C09065=1103.745,273.305,-76.182,179.309,15.397,151.389
C09066=1103.739,273.056,-76.153,179.306,15.397,151.390
C09067=1103.734,272.808,-76.125,179.302,15.395,151.390
C09068=1103.728,272.560,-76.096,179.298,15.395,151.391
C09069=1103.723,272.312,-76.068,179.294,15.394,151.392
C09070=1103.717,272.063,-76.039,179.291,15.393,151.392
C09071=1103.711,271.815,-76.010,179.287,15.393,151.393
C09072=1103.706,271.567,-75.982,179.283,15.392,151.394
C09073=1103.700,271.318,-75.954,179.280,15.391,151.394
C09074=1103.695,271.070,-75.925,179.276,15.390,151.395
C09075=1103.689,270.822,-75.897,179.272,15.390,151.395
C09076=1103.683,270.574,-75.869,179.269,15.389,151.396
C09077=1103.677,270.325,-75.840,179.265,15.388,151.397
C09078=1103.671,270.077,-75.811,179.262,15.387,151.397
C09079=1103.666,269.829,-75.783,179.257,15.386,151.398
C09080=1103.660,269.580,-75.755,179.254,15.386,151.399
C09081=1103.655,269.332,-75.727,179.250,15.385,151.399
C09082=1103.649,269.083,-75.699,179.246,15.384,151.400
C09083=1103.644,268.835,-75.669,179.243,15.384,151.400
C09084=1103.638,268.587,-75.641,179.239,15.383,151.401
C09085=1103.632,268.339,-75.613,179.235,15.382,151.402
C09086=1103.626,268.090,-75.585,179.232,15.382,151.402
C09087=1103.621,267.842,-75.557,179.228,15.381,151.403
C09088=1103.615,267.593,-75.528,179.224,15.380,151.404
C09089=1103.610,267.345,-75.501,179.220,15.379,151.404
C09090=1103.604,267.097,-75.471,179.217,15.379,151.405
C09091=1103.598,266.849,-75.444,179.213,15.378,151.405
C09092=1103.592,266.600,-75.415,179.209,15.377,151.406
C09093=1103.587,266.352,-75.387,179.206,15.377,151.407
C09094=1103.581,266.103,-75.359,179.202,15.376,151.407
C09095=1103.576,265.855,-75.331,179.198,15.375,151.408
C09096=1103.570,265.606,-75.303,179.195,15.375,151.409
C09097=1103.564,265.358,-75.275,179.191,15.374,151.409
C09098=1103.558,265.110,-75.246,179.187,15.373,151.410
C09099=1103.552,264.862,-75.219,179.184,15.373,151.411
C09100=1103.547,264.614,-75.191,179.179,15.372,151.411
C09101=1103.541,264.365,-75.163,179.176,15.371,151.412
C09102=1103.536,264.117,-75.135,179.173,15.371,151.412
C09103=1103.530,263.868,-75.107,179.168,15.370,151.413
C09104=1103.525,263.620,-75.079,179.165,15.370,151.414
C09105=1103.516,263.267,-75.039,179.160,15.368,151.415
C09106=1103.507,262.913,-74.999,179.155,15.368,151.416
C09107=1103.499,262.559,-74.960,179.149,15.367,151.417
C09108=1103.491,262.206,-74.920,179.144,15.366,151.418
C09109=1103.486,261.957,-74.893,179.140,15.366,151.418
C09110=1103.480,261.708,-74.865,179.136,15.365,151.419
C09111=1103.475,261.460,-74.837,179.133,15.364,151.420
C09112=1103.468,261.212,-74.809,179.129,15.364,151.420
C09113=1103.463,260.964,-74.781,179.125,15.363,151.421
C09114=1103.458,260.715,-74.754,179.121,15.363,151.422
C09115=1103.451,260.467,-74.726,179.118,15.363,151.422
C09116=1103.445,260.219,-74.698,179.114,15.361,151.423
C09117=1103.440,259.970,-74.670,179.110,15.361,151.424
C09118=1103.434,259.721,-74.643,179.107,15.361,151.424
C09119=1103.428,259.473,-74.615,179.102,15.360,151.425
C09120=1103.422,259.225,-74.587,179.099,15.359,151.426
C09121=1103.417,258.976,-74.560,179.095,15.359,151.426
C09122=1103.411,258.728,-74.532,179.092,15.359,151.427
C09123=1103.405,258.480,-74.504,179.088,15.358,151.428
C09124=1103.400,258.231,-74.477,179.084,15.357,151.428
C09125=1103.394,257.982,-74.449,179.081,15.357,151.429
C09126=1103.389,257.734,-74.422,179.077,15.356,151.430
C09127=1103.383,257.486,-74.394,179.073,15.356,151.430
C09128=1103.377,257.237,-74.366,179.069,15.355,151.431
C09129=1103.371,256.989,-74.339,179.065,15.355,151.432
C09130=1103.366,256.741,-74.311,179.062,15.354,151.432
C09131=1103.360,256.492,-74.284,179.058,15.354,151.433
C09132=1103.354,256.244,-74.256,179.054,15.353,151.434
C09133=1103.349,255.995,-74.229,179.051,15.352,151.434
C09134=1103.343,255.747,-74.202,179.047,15.352,151.435
C09135=1103.337,255.498,-74.174,179.044,15.352,151.436
C09136=1103.332,255.250,-74.146,179.039,15.351,151.436
C09137=1103.326,255.002,-74.119,179.036,15.351,151.437
C09138=1103.321,254.753,-74.092,179.033,15.350,151.438
C09139=1103.314,254.504,-74.065,179.028,15.349,151.438
C09140=1103.309,254.256,-74.037,179.025,15.349,151.439
C09141=1103.303,254.008,-74.010,179.021,15.348,151.440
C09142=1103.298,253.759,-73.983,179.017,15.348,151.440
C09143=1103.292,253.510,-73.956,179.013,15.347,151.441
C09144=1103.286,253.262,-73.928,179.010,15.347,151.442
C09145=1103.281,253.014,-73.901,179.006,15.347,151.443
C09146=1103.276,252.765,-73.874,179.002,15.345,151.443
C09147=1103.269,252.517,-73.846,178.999,15.345,151.444
C09148=1103.264,252.268,-73.819,178.995,15.345,151.445
C09149=1103.258,252.020,-73.792,178.991,15.344,151.445
C09150=1103.253,251.772,-73.764,178.987,15.344,151.446
C09151=1103.247,251.523,-73.738,178.984,15.343,151.447
C09152=1103.242,251.275,-73.710,178.980,15.343,151.447
C09153=1103.236,251.026,-73.684,178.976,15.342,151.448
C09154=1103.230,250.778,-73.655,178.973,15.342,151.449
C09155=1103.224,250.529,-73.629,178.969,15.341,151.449
C09156=1103.219,250.280,-73.601,178.966,15.341,151.450
C09157=1103.211,249.924,-73.563,178.960,15.340,151.451
C09158=1103.203,249.568,-73.524,178.954,15.339,151.452
C09159=1103.195,249.212,-73.485,178.949,15.338,151.453
C09160=1103.187,248.854,-73.446,178.944,15.338,151.454
C09161=1103.182,248.606,-73.420,178.940,15.337,151.455
C09162=1103.176,248.358,-73.393,178.937,15.337,151.455
C09163=1103.171,248.110,-73.365,178.933,15.336,151.456
C09164=1103.165,247.861,-73.338,178.930,15.336,151.457
C09165=1103.160,247.613,-73.311,178.925,15.335,151.457
C09166=1103.154,247.364,-73.284,178.922,15.335,151.458
C09167=1103.148,247.116,-73.258,178.918,15.335,151.459
C09168=1103.142,246.868,-73.231,178.915,15.334,151.459
C09169=1103.137,246.619,-73.204,178.910,15.334,151.460
C09170=1103.131,246.370,-73.177,178.907,15.333,151.461
C09171=1103.125,246.121,-73.150,178.903,15.333,151.462
C09172=1103.120,245.873,-73.124,178.900,15.333,151.462
C09173=1103.114,245.624,-73.096,178.896,15.332,151.463
C09174=1103.109,245.376,-73.070,178.892,15.332,151.464
C09175=1103.103,245.128,-73.043,178.888,15.331,151.464
C09176=1103.097,244.879,-73.017,178.885,15.331,151.465
C09177=1103.092,244.630,-72.990,178.881,15.331,151.466
C09178=1103.087,244.382,-72.963,178.877,15.330,151.466
C09179=1103.081,244.133,-72.937,178.874,15.330,151.467
C09180=1103.075,243.885,-72.910,178.870,15.329,151.468
C09181=1103.069,243.637,-72.883,178.867,15.329,151.469
C09182=1103.064,243.388,-72.856,178.862,15.328,151.469
C09183=1103.059,243.139,-72.830,178.859,15.328,151.470
C09184=1103.053,242.891,-72.804,178.855,15.328,151.471
C09185=1103.046,242.576,-72.770,178.851,15.327,151.472
C09186=1103.038,242.261,-72.736,178.846,15.327,151.473
C09187=1103.031,241.946,-72.703,178.841,15.327,151.473
C09188=1103.023,241.631,-72.669,178.836,15.326,151.474
C09189=1103.018,241.382,-72.643,178.832,15.325,151.475
C09190=1103.012,241.133,-72.616,178.829,15.325,151.476
C09191=1103.006,240.885,-72.589,178.825,15.325,151.476
C09192=1103.001,240.637,-72.563,178.821,15.325,151.477
C09193=1102.996,240.387,-72.536,178.818,15.324,151.478
C09194=1102.990,240.139,-72.510,178.813,15.324,151.479
C09195=1102.984,239.891,-72.483,178.810,15.324,151.479
C09196=1102.978,239.642,-72.458,178.806,15.323,151.480
C09197=1102.972,239.394,-72.431,178.803,15.323,151.481
C09198=1102.966,239.145,-72.404,178.799,15.323,151.482
C09199=1102.961,238.896,-72.378,178.795,15.322,151.482
C09200=1102.955,238.648,-72.352,178.791,15.322,151.483
C09201=1102.950,238.399,-72.326,178.788,15.321,151.484
C09202=1102.944,238.151,-72.299,178.784,15.321,151.484
C09203=1102.938,237.902,-72.273,178.780,15.321,151.485
C09204=1102.933,237.653,-72.247,178.777,15.321,151.486
C09205=1102.927,237.405,-72.220,178.773,15.320,151.487
C09206=1102.922,237.157,-72.194,178.769,15.320,151.487
C09207=1102.916,236.908,-72.168,178.766,15.320,151.488
C09208=1102.911,236.659,-72.142,178.762,15.320,151.489
C09209=1102.904,236.362,-72.111,178.757,15.319,151.490
C09210=1102.896,236.066,-72.079,178.753,15.319,151.491
C09211=1102.891,235.769,-72.048,178.748,15.318,151.491
C09212=1102.884,235.472,-72.017,178.744,15.318,151.492
C09213=1102.878,235.224,-71.990,178.740,15.317,151.493
C09214=1102.872,234.975,-71.964,178.736,15.317,151.494
C09215=1102.867,234.727,-71.939,178.733,15.317,151.494
C09216=1102.861,234.479,-71.913,178.729,15.317,151.495
C09217=1102.856,234.230,-71.887,178.726,15.316,151.496
C09218=1102.850,233.981,-71.861,178.722,15.317,151.497
C09219=1102.844,233.732,-71.834,178.718,15.316,151.497
C09220=1102.839,233.483,-71.808,178.714,15.316,151.498
C09221=1102.833,233.235,-71.783,178.711,15.315,151.499
C09222=1102.827,232.987,-71.757,178.707,15.315,151.500
C09223=1102.822,232.738,-71.731,178.704,15.315,151.500
C09224=1102.817,232.489,-71.705,178.700,15.315,151.501
C09225=1102.810,232.241,-71.679,178.695,15.314,151.502
C09226=1102.805,231.992,-71.653,178.692,15.314,151.503
C09227=1102.799,231.743,-71.627,178.688,15.314,151.503
C09228=1102.794,231.495,-71.601,178.685,15.313,151.504
C09229=1102.788,231.247,-71.575,178.681,15.313,151.505
C09230=1102.782,230.998,-71.549,178.678,15.313,151.505
C09231=1102.777,230.749,-71.523,178.674,15.313,151.506
C09232=1102.771,230.500,-71.498,178.670,15.312,151.507
C09233=1102.766,230.252,-71.472,178.666,15.312,151.508
C09234=1102.760,230.003,-71.446,178.662,15.312,151.508
C09235=1102.754,229.755,-71.420,178.659,15.312,151.509
C09236=1102.748,229.506,-71.394,178.655,15.312,151.510
C09237=1102.742,229.257,-71.369,178.651,15.312,151.511
C09238=1102.737,229.009,-71.344,178.648,15.311,151.511
C09239=1102.732,228.760,-71.318,178.644,15.311,151.512
C09240=1102.725,228.511,-71.292,178.640,15.311,151.513
C09241=1102.720,228.262,-71.266,178.636,15.310,151.514
C09242=1102.714,228.013,-71.241,178.633,15.310,151.514
C09243=1102.709,227.765,-71.215,178.629,15.310,151.515
C09244=1102.703,227.517,-71.190,178.625,15.310,151.516
C09245=1102.697,227.268,-71.164,178.622,15.310,151.517
C09246=1102.691,227.019,-71.139,178.618,15.310,151.517
C09247=1102.686,226.771,-71.113,178.615,15.310,151.518
C09248=1102.680,226.522,-71.088,178.610,15.309,151.519
C09249=1102.675,226.273,-71.062,178.607,15.309,151.520
C09250=1102.669,226.025,-71.037,178.603,15.309,151.520
C09251=1102.663,225.776,-71.011,178.599,15.308,151.521
C09252=1102.657,225.527,-70.986,178.596,15.308,151.522
C09253=1102.652,225.278,-70.960,178.592,15.308,151.523
C09254=1102.646,225.030,-70.935,178.588,15.308,151.523
C09255=1102.641,224.781,-70.909,178.585,15.308,151.524
C09256=1102.634,224.533,-70.884,178.581,15.308,151.525
C09257=1102.630,224.284,-70.858,178.577,15.307,151.526
C09258=1102.623,224.036,-70.833,178.573,15.307,151.527
C09259=1102.618,223.787,-70.807,178.570,15.307,151.527
C09260=1102.613,223.538,-70.783,178.566,15.307,151.528
C09261=1102.604,223.166,-70.744,178.560,15.306,151.529
C09262=1102.596,222.795,-70.706,178.555,15.306,151.530
C09263=1102.587,222.424,-70.669,178.550,15.306,151.531
C09264=1102.579,222.051,-70.631,178.545,15.306,151.532
C09265=1102.574,221.803,-70.606,178.540,15.305,151.533
C09266=1102.567,221.555,-70.580,178.536,15.305,151.534
C09267=1102.562,221.305,-70.555,178.533,15.305,151.535
C09268=1102.557,221.057,-70.530,178.529,15.305,151.535
C09269=1102.550,220.809,-70.505,178.525,15.305,151.536
C09270=1102.545,220.560,-70.479,178.522,15.305,151.537
C09271=1102.540,220.311,-70.455,178.518,15.304,151.538
C09272=1102.533,220.062,-70.429,178.514,15.305,151.539
C09273=1102.527,219.814,-70.404,178.511,15.305,151.539
C09274=1102.523,219.565,-70.379,178.507,15.304,151.540
C09275=1102.516,219.316,-70.354,178.504,15.304,151.541
C09276=1102.511,219.068,-70.330,178.500,15.304,151.542
C09277=1102.505,218.819,-70.304,178.496,15.304,151.542
C09278=1102.499,218.570,-70.278,178.493,15.304,151.543
C09279=1102.494,218.321,-70.254,178.488,15.303,151.544
C09280=1102.488,218.073,-70.229,178.485,15.303,151.545
C09281=1102.483,217.824,-70.204,178.481,15.303,151.545
C09282=1102.476,217.575,-70.179,178.478,15.303,151.546
C09283=1102.472,217.326,-70.154,178.474,15.303,151.547
C09284=1102.466,217.078,-70.129,178.470,15.303,151.548
C09285=1102.460,216.829,-70.105,178.467,15.303,151.548
C09286=1102.454,216.581,-70.079,178.463,15.303,151.549
C09287=1102.449,216.332,-70.055,178.459,15.303,151.550
C09288=1102.443,216.083,-70.029,178.456,15.302,151.551
C09289=1102.438,215.834,-70.005,178.452,15.302,151.551
C09290=1102.432,215.586,-69.979,178.448,15.302,151.552
C09291=1102.427,215.337,-69.955,178.445,15.302,151.553
C09292=1102.420,215.088,-69.930,178.441,15.302,151.554
C09293=1102.415,214.840,-69.906,178.438,15.302,151.554
C09294=1102.409,214.591,-69.880,178.434,15.302,151.555
C09295=1102.404,214.342,-69.855,178.430,15.302,151.556
C09296=1102.398,214.093,-69.831,178.426,15.301,151.557
C09297=1102.393,213.845,-69.806,178.422,15.301,151.558
C09298=1102.387,213.596,-69.781,178.419,15.301,151.558
C09299=1102.382,213.347,-69.757,178.415,15.301,151.559
C09300=1102.375,213.098,-69.732,178.411,15.301,151.560
C09301=1102.370,212.850,-69.707,178.408,15.301,151.561
C09302=1102.364,212.601,-69.683,178.404,15.301,151.561
C09303=1102.359,212.353,-69.658,178.400,15.301,151.562
C09304=1102.353,212.103,-69.633,178.397,15.301,151.563
C09305=1102.347,211.855,-69.609,178.393,15.301,151.564
C09306=1102.342,211.606,-69.585,178.390,15.300,151.564
C09307=1102.336,211.358,-69.559,178.386,15.301,151.565
C09308=1102.331,211.109,-69.535,178.382,15.300,151.566
C09309=1102.325,210.860,-69.510,178.379,15.300,151.567
C09310=1102.319,210.611,-69.486,178.375,15.300,151.568
C09311=1102.313,210.362,-69.461,178.371,15.300,151.568
C09312=1102.308,210.114,-69.437,178.368,15.300,151.569
C09313=1102.299,209.746,-69.401,178.362,15.300,151.570
C09314=1102.291,209.378,-69.364,178.357,15.300,151.571
C09315=1102.283,209.010,-69.329,178.352,15.300,151.572
C09316=1102.274,208.642,-69.292,178.346,15.300,151.574
C09317=1102.252,207.639,-69.194,178.312,15.293,151.579
C09318=1102.246,207.391,-69.170,178.308,15.294,151.580
C09319=1102.240,207.142,-69.146,178.304,15.294,151.581
C09320=1102.234,206.893,-69.122,178.301,15.296,151.582
C09321=1102.229,206.644,-69.097,178.297,15.296,151.583
C09322=1102.222,206.395,-69.073,178.292,15.297,151.585
C09323=1102.217,206.147,-69.049,178.289,15.297,151.585
C09324=1102.212,205.898,-69.025,178.285,15.299,151.586
C09325=1102.206,205.648,-69.001,178.281,15.299,151.587
C09326=1102.200,205.400,-68.977,178.277,15.300,151.589
C09327=1102.195,205.151,-68.953,178.274,15.301,151.589
C09328=1102.190,204.903,-68.929,178.269,15.302,151.590
C09329=1102.183,204.654,-68.905,178.265,15.302,151.591
C09330=1102.178,204.405,-68.880,178.261,15.303,151.593
C09331=1102.172,204.157,-68.856,178.258,15.304,151.593
C09332=1102.167,203.908,-68.833,178.254,15.305,151.594
C09333=1102.161,203.659,-68.809,178.250,15.305,151.596
C09334=1102.155,203.410,-68.784,178.246,15.305,151.596
C09335=1102.149,203.162,-68.761,178.242,15.307,151.597
C09336=1102.144,202.913,-68.736,178.238,15.307,151.598
C09337=1102.139,202.663,-68.712,178.234,15.308,151.600
C09338=1102.132,202.415,-68.689,178.231,15.309,151.600
C09339=1102.127,202.166,-68.665,178.227,15.310,151.601
C09340=1102.121,201.917,-68.641,178.222,15.310,151.603
C09341=1102.116,201.668,-68.617,178.218,15.311,151.604
C09342=1102.110,201.420,-68.593,178.215,15.312,151.604
C09343=1102.104,201.171,-68.569,178.211,15.313,151.605
C09344=1102.098,200.922,-68.545,178.207,15.314,151.607
C09345=1102.093,200.673,-68.521,178.203,15.315,151.608
C09346=1102.087,200.425,-68.498,178.200,15.315,151.608
C09347=1102.081,200.177,-68.474,178.195,15.316,151.610
C09348=1102.075,199.927,-68.450,178.191,15.317,151.611
C09349=1102.069,199.678,-68.427,178.188,15.317,151.611
C09350=1102.064,199.430,-68.402,178.184,15.318,151.612
C09351=1102.058,199.181,-68.379,178.180,15.319,151.614
C09352=1102.052,198.932,-68.355,178.177,15.320,151.614
C09353=1102.046,198.683,-68.332,178.172,15.320,151.615
C09354=1102.041,198.434,-68.308,178.168,15.321,151.617
C09355=1102.035,198.185,-68.285,178.165,15.322,151.617
C09356=1102.029,197.937,-68.261,178.161,15.323,151.618
C09357=1102.023,197.688,-68.236,178.157,15.323,151.620
C09358=1102.018,197.439,-68.213,178.153,15.324,151.620
C09359=1102.012,197.190,-68.189,178.149,15.325,151.621
C09360=1102.006,196.941,-68.166,178.146,15.325,151.622
C09361=1102.000,196.693,-68.143,178.141,15.326,151.623
C09362=1101.995,196.444,-68.119,178.138,15.327,151.624
C09363=1101.989,196.195,-68.095,178.134,15.328,151.625
C09364=1101.983,195.946,-68.072,178.130,15.328,151.626
C09365=1101.978,195.697,-68.048,178.127,15.329,151.627
C09366=1101.972,195.448,-68.025,178.123,15.330,151.628
C09367=1101.966,195.199,-68.002,178.119,15.330,151.629
C09368=1101.961,194.951,-67.978,178.115,15.331,151.630
C09369=1101.955,194.702,-67.955,178.111,15.332,151.631
C09370=1101.949,194.454,-67.931,178.107,15.333,151.632
C09371=1101.944,194.204,-67.907,178.103,15.333,151.633
C09372=1101.938,193.955,-67.884,178.100,15.334,151.634
C09373=1101.932,193.707,-67.860,178.096,15.335,151.635
C09374=1101.927,193.457,-67.837,178.092,15.335,151.636
C09375=1101.921,193.209,-67.814,178.089,15.336,151.637
C09376=1101.915,192.960,-67.790,178.085,15.337,151.638
C09377=1101.910,192.711,-67.767,178.081,15.337,151.639
C09378=1101.904,192.439,-67.742,178.077,15.338,151.640
C09379=1101.897,192.167,-67.715,178.072,15.339,151.641
C09380=1101.892,191.894,-67.690,178.068,15.339,151.642
C09381=1101.885,191.621,-67.665,178.064,15.340,151.643
C09382=1101.879,191.373,-67.642,178.061,15.342,151.644
C09383=1101.874,191.123,-67.618,178.057,15.342,151.645
C09384=1101.868,190.875,-67.595,178.053,15.342,151.646
C09385=1101.862,190.626,-67.572,178.049,15.344,151.647
C09386=1101.857,190.377,-67.549,178.046,15.344,151.648
C09387=1101.852,190.128,-67.525,178.041,15.345,151.649
C09388=1101.846,189.879,-67.502,178.037,15.345,151.650
C09389=1101.840,189.631,-67.479,178.034,15.346,151.651
C09390=1101.834,189.382,-67.456,178.030,15.346,151.652
C09391=1101.829,189.133,-67.432,178.026,15.347,151.653
C09392=1101.823,188.884,-67.409,178.023,15.348,151.653
C09393=1101.818,188.635,-67.386,178.019,15.348,151.655
C09394=1101.812,188.386,-67.363,178.015,15.349,151.655
C09395=1101.807,188.138,-67.341,178.012,15.350,151.656
C09396=1101.802,187.889,-67.317,178.008,15.350,151.657
C09397=1101.796,187.640,-67.294,178.004,15.351,151.658
C09398=1101.790,187.392,-67.271,178.001,15.352,151.659
C09399=1101.784,187.143,-67.248,177.997,15.352,151.660
C09400=1101.779,186.894,-67.225,177.993,15.353,151.661
C09401=1101.774,186.645,-67.201,177.989,15.353,151.662
C09402=1101.768,186.396,-67.178,177.986,15.354,151.663
C09403=1101.762,186.147,-67.155,177.982,15.354,151.664
C09404=1101.756,185.898,-67.132,177.978,15.355,151.665
C09405=1101.751,185.649,-67.109,177.975,15.356,151.666
C09406=1101.746,185.401,-67.087,177.971,15.356,151.667
C09407=1101.740,185.152,-67.064,177.967,15.357,151.667
C09408=1101.734,184.902,-67.042,177.963,15.358,151.668
C09409=1101.729,184.653,-67.019,177.960,15.358,151.669
C09410=1101.723,184.405,-66.996,177.956,15.358,151.670
C09411=1101.717,184.156,-66.973,177.952,15.360,151.671
C09412=1101.712,183.907,-66.950,177.948,15.360,151.672
C09413=1101.706,183.658,-66.927,177.945,15.360,151.673
C09414=1101.700,183.409,-66.904,177.941,15.362,151.674
C09415=1101.694,183.160,-66.882,177.937,15.362,151.675
C09416=1101.688,182.912,-66.859,177.933,15.362,151.676
C09417=1101.682,182.663,-66.836,177.930,15.364,151.677
C09418=1101.676,182.414,-66.813,177.926,15.364,151.678
C09419=1101.671,182.164,-66.791,177.922,15.364,151.679
C09420=1101.665,181.915,-66.768,177.919,15.366,151.680
C09421=1101.659,181.667,-66.745,177.915,15.366,151.681
C09422=1101.653,181.418,-66.722,177.911,15.367,151.682
C09423=1101.647,181.169,-66.699,177.908,15.367,151.682
C09424=1101.642,180.919,-66.677,177.904,15.368,151.684
C09425=1101.636,180.670,-66.654,177.900,15.369,151.684
C09426=1101.630,180.423,-66.632,177.897,15.369,151.685
C09427=1101.625,180.174,-66.609,177.893,15.370,151.686
C09428=1101.619,179.924,-66.587,177.889,15.371,151.687
C09429=1101.613,179.675,-66.564,177.886,15.371,151.688
C09430=1101.608,179.426,-66.541,177.882,15.372,151.689
C09431=1101.601,179.178,-66.519,177.878,15.372,151.690
C09432=1101.596,178.928,-66.497,177.875,15.373,151.691
C09433=1101.590,178.679,-66.474,177.871,15.374,151.692
C09434=1101.585,178.431,-66.451,177.867,15.374,151.693
C09435=1101.579,178.182,-66.429,177.864,15.375,151.694
C09436=1101.573,177.933,-66.406,177.860,15.375,151.695
C09437=1101.567,177.684,-66.384,177.856,15.376,151.695
C09438=1101.562,177.435,-66.361,177.853,15.377,151.696
C09439=1101.555,177.186,-66.339,177.849,15.377,151.697
C09440=1101.551,176.937,-66.317,177.845,15.378,151.698
C09441=1101.545,176.688,-66.294,177.842,15.379,151.699
C09442=1101.539,176.415,-66.270,177.838,15.379,151.700
C09443=1101.532,176.143,-66.245,177.833,15.380,151.701
C09444=1101.526,175.870,-66.221,177.830,15.380,151.702
C09445=1101.519,175.597,-66.196,177.825,15.381,151.703
C09446=1101.514,175.349,-66.174,177.822,15.382,151.704
C09447=1101.509,175.099,-66.151,177.818,15.382,151.705
C09448=1101.502,174.851,-66.129,177.815,15.383,151.706
C09449=1101.497,174.601,-66.107,177.811,15.384,151.707
C09450=1101.492,174.353,-66.084,177.808,15.384,151.707
C09451=1101.486,174.104,-66.063,177.804,15.384,151.708
C09452=1101.480,173.855,-66.040,177.801,15.385,151.709
C09453=1101.474,173.605,-66.017,177.797,15.385,151.710
C09454=1101.469,173.357,-65.995,177.793,15.386,151.711
C09455=1101.463,173.108,-65.973,177.790,15.387,151.712
C09456=1101.457,172.859,-65.952,177.786,15.387,151.713
C09457=1101.452,172.611,-65.929,177.782,15.387,151.714
C09458=1101.446,172.361,-65.907,177.779,15.388,151.715
C09459=1101.440,172.112,-65.884,177.775,15.389,151.715
C09460=1101.435,171.863,-65.862,177.771,15.389,151.716
C09461=1101.430,171.614,-65.840,177.768,15.390,151.717
C09462=1101.423,171.366,-65.818,177.764,15.390,151.718
C09463=1101.418,171.116,-65.796,177.761,15.390,151.719
C09464=1101.412,170.867,-65.775,177.757,15.391,151.720
C09465=1101.407,170.619,-65.752,177.754,15.392,151.721
C09466=1101.401,170.369,-65.729,177.750,15.392,151.722
C09467=1101.396,170.121,-65.708,177.747,15.393,151.722
C09468=1101.390,169.872,-65.685,177.743,15.393,151.723
C09469=1101.384,169.622,-65.663,177.740,15.394,151.724
C09470=1101.379,169.374,-65.642,177.736,15.394,151.725
C09471=1101.373,169.124,-65.620,177.732,15.394,151.726
C09472=1101.368,168.876,-65.597,177.729,15.395,151.727
C09473=1101.362,168.627,-65.575,177.725,15.396,151.728
C09474=1101.356,168.378,-65.554,177.721,15.396,151.729
C09475=1101.351,168.129,-65.532,177.718,15.397,151.729
C09476=1101.345,167.880,-65.510,177.715,15.397,151.730
C09477=1101.340,167.631,-65.487,177.711,15.397,151.731
C09478=1101.334,167.382,-65.466,177.708,15.398,151.732
C09479=1101.328,167.133,-65.444,177.704,15.398,151.733
C09480=1101.323,166.884,-65.422,177.700,15.398,151.734
C09481=1101.317,166.635,-65.400,177.697,15.399,151.734
C09482=1101.312,166.386,-65.379,177.693,15.400,151.735
C09483=1101.306,166.137,-65.357,177.690,15.400,151.736
C09484=1101.301,165.888,-65.335,177.687,15.401,151.737
C09485=1101.295,165.639,-65.312,177.683,15.401,151.738
C09486=1101.289,165.391,-65.291,177.680,15.402,151.739
C09487=1101.284,165.141,-65.269,177.676,15.402,151.739
C09488=1101.278,164.893,-65.248,177.672,15.402,151.740
C09489=1101.273,164.643,-65.225,177.669,15.403,151.741
C09490=1101.267,164.394,-65.204,177.665,15.403,151.742
C09491=1101.262,164.145,-65.182,177.662,15.403,151.743
C09492=1101.256,163.896,-65.160,177.659,15.404,151.744
C09493=1101.251,163.647,-65.138,177.655,15.404,151.745
C09494=1101.245,163.399,-65.117,177.651,15.405,151.745
C09495=1101.239,163.149,-65.095,177.648,15.405,151.746
C09496=1101.235,162.901,-65.074,177.644,15.406,151.747
C09497=1101.228,162.651,-65.052,177.641,15.406,151.748
C09498=1101.224,162.403,-65.030,177.638,15.406,151.749
C09499=1101.217,162.153,-65.008,177.634,15.406,151.749
C09500=1101.213,161.905,-64.987,177.631,15.407,151.750
C09501=1101.207,161.655,-64.966,177.627,15.408,151.751
C09502=1101.201,161.406,-64.944,177.624,15.408,151.752
C09503=1101.195,161.157,-64.923,177.620,15.409,151.753
C09504=1101.190,160.908,-64.901,177.617,15.409,151.754
C09505=1101.184,160.659,-64.879,177.613,15.409,151.754
C09506=1101.178,160.385,-64.856,177.610,15.410,151.755
C09507=1101.172,160.113,-64.832,177.606,15.410,151.756
C09508=1101.166,159.840,-64.809,177.602,15.411,151.757
C09509=1101.159,159.567,-64.785,177.598,15.411,151.758
C09510=1101.154,159.318,-64.764,177.594,15.411,151.759
C09511=1101.148,159.068,-64.742,177.591,15.412,151.760
C09512=1101.142,158.820,-64.721,177.588,15.412,151.761
C09513=1101.136,158.571,-64.699,177.584,15.413,151.761
C09514=1101.131,158.322,-64.678,177.581,15.413,151.762
C09515=1101.125,158.072,-64.657,177.577,15.413,151.763
C09516=1101.120,157.823,-64.635,177.574,15.414,151.764
C09517=1101.114,157.574,-64.614,177.570,15.414,151.765
C09518=1101.108,157.326,-64.592,177.567,15.414,151.765
C09519=1101.102,157.076,-64.572,177.564,15.415,151.766
C09520=1101.097,156.827,-64.550,177.560,15.415,151.767
C09521=1101.091,156.579,-64.529,177.556,15.416,151.768
C09522=1101.085,156.329,-64.508,177.554,15.416,151.769
C09523=1101.080,156.080,-64.486,177.550,15.417,151.770
C09524=1101.074,155.831,-64.465,177.547,15.417,151.770
C09525=1101.069,155.582,-64.444,177.543,15.417,151.771
C09526=1101.064,155.333,-64.423,177.539,15.417,151.772
C09527=1101.057,155.084,-64.401,177.536,15.418,151.773
C09528=1101.052,154.835,-64.381,177.533,15.418,151.774
C09529=1101.046,154.586,-64.359,177.530,15.419,151.774
C09530=1101.040,154.337,-64.338,177.526,15.419,151.775
C09531=1101.035,154.088,-64.317,177.522,15.420,151.776
C09532=1101.029,153.839,-64.295,177.519,15.420,151.777
C09533=1101.024,153.590,-64.275,177.515,15.420,151.778
C09534=1101.018,153.341,-64.253,177.512,15.420,151.778
C09535=1101.012,153.092,-64.232,177.509,15.421,151.779
C09536=1101.007,152.843,-64.211,177.505,15.421,151.780
C09537=1101.001,152.594,-64.190,177.502,15.422,151.781
C09538=1100.995,152.345,-64.169,177.499,15.422,151.782
C09539=1100.989,152.096,-64.148,177.495,15.422,151.782
C09540=1100.984,151.846,-64.127,177.492,15.423,151.783
C09541=1100.978,151.598,-64.106,177.488,15.423,151.784
C09542=1100.972,151.348,-64.085,177.486,15.424,151.785
C09543=1100.967,151.100,-64.064,177.482,15.424,151.786
C09544=1100.962,150.851,-64.043,177.478,15.424,151.786
C09545=1100.955,150.601,-64.021,177.475,15.425,151.787
C09546=1100.950,150.352,-64.001,177.472,15.424,151.788
C09547=1100.945,150.103,-63.980,177.469,15.425,151.789
C09548=1100.939,149.854,-63.959,177.465,15.425,151.790
C09549=1100.933,149.605,-63.939,177.461,15.425,151.790
C09550=1100.927,149.357,-63.917,177.459,15.426,151.791
C09551=1100.922,149.107,-63.897,177.455,15.426,151.792
C09552=1100.916,148.858,-63.876,177.452,15.427,151.793
C09553=1100.911,148.609,-63.855,177.448,15.427,151.793
C09554=1100.905,148.360,-63.834,177.445,15.427,151.794
C09555=1100.899,148.110,-63.813,177.442,15.428,151.795
C09556=1100.894,147.862,-63.792,177.438,15.428,151.796
C09557=1100.888,147.613,-63.772,177.435,15.428,151.796
C09558=1100.882,147.363,-63.751,177.431,15.429,151.797
C09559=1100.876,147.114,-63.730,177.428,15.429,151.798
C09560=1100.871,146.865,-63.709,177.425,15.429,151.799
C09561=1100.865,146.617,-63.689,177.422,15.429,151.800
C09562=1100.859,146.367,-63.668,177.418,15.430,151.800
C09563=1100.854,146.118,-63.647,177.415,15.430,151.801
C09564=1100.849,145.869,-63.627,177.411,15.430,151.802
C09565=1100.842,145.620,-63.606,177.408,15.430,151.803
C09566=1100.836,145.371,-63.585,177.405,15.430,151.803
C09567=1100.831,145.122,-63.564,177.402,15.431,151.804
C09568=1100.826,144.873,-63.544,177.398,15.431,151.805
C09569=1100.820,144.624,-63.524,177.395,15.431,151.806
C09570=1100.814,144.350,-63.500,177.392,15.432,151.807
C09571=1100.807,144.076,-63.478,177.388,15.432,151.807
C09572=1100.801,143.804,-63.455,177.384,15.433,151.808
C09573=1100.795,143.530,-63.433,177.381,15.433,151.809
C09574=1100.789,143.281,-63.412,177.377,15.433,151.810
C09575=1100.784,143.032,-63.391,177.374,15.433,151.810
C09576=1100.778,142.783,-63.371,177.371,15.433,151.811
C09577=1100.772,142.534,-63.351,177.368,15.434,151.812
C09578=1100.767,142.284,-63.330,177.364,15.434,151.813
C09579=1100.761,142.036,-63.310,177.361,15.435,151.814
C09580=1100.756,141.787,-63.289,177.358,15.434,151.814
C09581=1100.751,141.537,-63.269,177.354,15.434,151.815
C09582=1100.745,141.289,-63.249,177.351,15.435,151.816
C09583=1100.739,141.039,-63.228,177.348,15.435,151.817
C09584=1100.733,140.790,-63.207,177.345,15.436,151.817
C09585=1100.727,140.541,-63.187,177.341,15.435,151.818
C09586=1100.722,140.292,-63.166,177.338,15.435,151.819
C09587=1100.716,140.044,-63.146,177.335,15.436,151.819
C09588=1100.711,139.794,-63.126,177.331,15.436,151.820
C09589=1100.705,139.545,-63.105,177.329,15.436,151.821
C09590=1100.699,139.295,-63.086,177.325,15.436,151.822
C09591=1100.694,139.046,-63.065,177.321,15.436,151.822
C09592=1100.688,138.797,-63.045,177.319,15.437,151.823
C09593=1100.683,138.548,-63.024,177.315,15.437,151.824
C09594=1100.677,138.299,-63.005,177.312,15.437,151.825
C09595=1100.671,138.050,-62.984,177.309,15.437,151.825
C09596=1100.665,137.801,-62.964,177.306,15.438,151.826
C09597=1100.659,137.551,-62.943,177.302,15.438,151.827
C09598=1100.653,137.303,-62.923,177.299,15.438,151.828
C09599=1100.648,137.054,-62.903,177.296,15.438,151.828
C09600=1100.642,136.805,-62.883,177.292,15.438,151.829
C09601=1100.637,136.556,-62.862,177.290,15.439,151.830
C09602=1100.631,136.306,-62.843,177.286,15.439,151.831
C09603=1100.626,136.057,-62.822,177.283,15.439,151.831
C09604=1100.620,135.808,-62.802,177.280,15.439,151.832
C09605=1100.614,135.558,-62.781,177.276,15.439,151.833
C09606=1100.608,135.310,-62.761,177.274,15.440,151.833
C09607=1100.603,135.060,-62.741,177.270,15.440,151.834
C09608=1100.597,134.811,-62.722,177.267,15.440,151.835
C09609=1100.592,134.562,-62.701,177.264,15.440,151.835
C09610=1100.586,134.313,-62.681,177.261,15.441,151.836
C09611=1100.580,134.064,-62.661,177.257,15.440,151.837
C09612=1100.575,133.815,-62.641,177.254,15.440,151.838
C09613=1100.569,133.566,-62.621,177.251,15.441,151.838
C09614=1100.564,133.317,-62.601,177.248,15.441,151.839
C09615=1100.558,133.068,-62.581,177.245,15.441,151.840
C09616=1100.552,132.818,-62.562,177.241,15.441,151.840
C09617=1100.547,132.569,-62.541,177.239,15.441,151.841
C09618=1100.541,132.320,-62.521,177.235,15.441,151.842
C09619=1100.536,132.071,-62.501,177.232,15.441,151.843
C09620=1100.530,131.822,-62.481,177.229,15.442,151.843
C09621=1100.524,131.573,-62.461,177.225,15.441,151.844
C09622=1100.518,131.324,-62.442,177.223,15.442,151.845
C09623=1100.513,131.074,-62.422,177.219,15.442,151.845
C09624=1100.506,130.825,-62.401,177.216,15.442,151.846
C09625=1100.501,130.576,-62.382,177.213,15.442,151.847
C09626=1100.495,130.327,-62.362,177.210,15.443,151.848
C09627=1100.489,130.078,-62.342,177.207,15.442,151.848
C09628=1100.484,129.828,-62.322,177.203,15.442,151.849
C09629=1100.478,129.579,-62.302,177.200,15.443,151.850
C09630=1100.472,129.330,-62.283,177.197,15.443,151.850
C09631=1100.466,129.081,-62.263,177.194,15.443,151.851
C09632=1100.460,128.832,-62.243,177.191,15.443,151.852
C09633=1100.455,128.583,-62.223,177.188,15.444,151.852
C09634=1100.449,128.310,-62.202,177.184,15.444,151.853
C09635=1100.443,128.036,-62.180,177.181,15.444,151.854
C09636=1100.436,127.763,-62.158,177.177,15.444,151.855
C09637=1100.430,127.489,-62.137,177.174,15.444,151.855
C09638=1100.424,127.240,-62.117,177.171,15.444,151.856
C09639=1100.418,126.991,-62.098,177.167,15.444,151.857
C09640=1100.413,126.741,-62.077,177.165,15.444,151.857
C09641=1100.407,126.492,-62.058,177.161,15.444,151.858
C09642=1100.401,126.243,-62.038,177.159,15.444,151.859
C09643=1100.396,125.994,-62.019,177.155,15.444,151.859
C09644=1100.390,125.745,-61.999,177.152,15.445,151.860
C09645=1100.384,125.496,-61.980,177.149,15.444,151.861
C09646=1100.378,125.246,-61.961,177.145,15.444,151.862
C09647=1100.372,124.997,-61.941,177.143,15.445,151.862
C09648=1100.367,124.748,-61.921,177.139,15.444,151.863
C09649=1100.361,124.499,-61.901,177.137,15.445,151.864
C09650=1100.356,124.250,-61.882,177.133,15.445,151.864
C09651=1100.351,124.001,-61.863,177.130,15.445,151.865
C09652=1100.345,123.752,-61.843,177.127,15.445,151.865
C09653=1100.339,123.502,-61.823,177.124,15.445,151.866
C09654=1100.333,123.253,-61.804,177.121,15.445,151.867
C09655=1100.327,123.004,-61.784,177.118,15.445,151.867
C09656=1100.322,122.755,-61.765,177.115,15.445,151.868
C09657=1100.316,122.505,-61.746,177.112,15.445,151.869
C09658=1100.312,122.256,-61.726,177.109,15.445,151.869
C09659=1100.306,122.007,-61.706,177.105,15.445,151.870
C09660=1100.300,121.758,-61.687,177.103,15.445,151.871
C09661=1100.294,121.509,-61.668,177.099,15.445,151.871
C09662=1100.288,121.260,-61.648,177.097,15.445,151.872
C09663=1100.283,121.010,-61.629,177.093,15.445,151.873
C09664=1100.277,120.761,-61.609,177.091,15.445,151.873
C09665=1100.272,120.512,-61.591,177.087,15.445,151.874
C09666=1100.266,120.263,-61.571,177.085,15.445,151.875
C09667=1100.260,120.014,-61.551,177.082,15.445,151.875
C09668=1100.254,119.764,-61.532,177.078,15.445,151.876
C09669=1100.249,119.515,-61.513,177.075,15.445,151.877
C09670=1100.244,119.266,-61.494,177.072,15.445,151.877
C09671=1100.238,119.017,-61.475,177.069,15.445,151.878
C09672=1100.232,118.767,-61.455,177.066,15.445,151.878
C09673=1100.226,118.519,-61.436,177.063,15.445,151.879
C09674=1100.221,118.270,-61.417,177.060,15.445,151.880
C09675=1100.216,118.020,-61.397,177.058,15.445,151.880
C09676=1100.210,117.771,-61.378,177.054,15.445,151.881
C09677=1100.204,117.522,-61.359,177.051,15.445,151.882
C09678=1100.198,117.272,-61.340,177.048,15.445,151.882
C09679=1100.193,117.023,-61.321,177.045,15.445,151.883
C09680=1100.188,116.774,-61.302,177.042,15.445,151.884
C09681=1100.182,116.525,-61.282,177.039,15.444,151.884
C09682=1100.177,116.276,-61.263,177.036,15.444,151.885
C09683=1100.171,116.026,-61.244,177.033,15.444,151.885
C09684=1100.166,115.777,-61.225,177.030,15.445,151.886
C09685=1100.160,115.528,-61.206,177.027,15.444,151.887
C09686=1100.155,115.279,-61.187,177.025,15.444,151.887
C09687=1100.149,115.029,-61.168,177.021,15.444,151.888
C09688=1100.143,114.780,-61.149,177.019,15.444,151.888
C09689=1100.138,114.531,-61.130,177.015,15.444,151.889
C09690=1100.132,114.282,-61.111,177.013,15.444,151.890
C09691=1100.126,114.033,-61.092,177.009,15.444,151.890
C09692=1100.120,113.783,-61.072,177.007,15.444,151.891
C09693=1100.115,113.534,-61.053,177.003,15.444,151.892
C09694=1100.109,113.285,-61.035,177.000,15.443,151.892
C09695=1100.103,113.036,-61.016,176.998,15.443,151.893
C09696=1100.098,112.786,-60.996,176.994,15.443,151.893
C09697=1100.092,112.538,-60.977,176.992,15.444,151.894
C09698=1100.086,112.264,-60.957,176.988,15.443,151.895
C09699=1100.080,111.991,-60.936,176.985,15.443,151.895
C09700=1100.074,111.717,-60.916,176.982,15.443,151.896
C09701=1100.067,111.444,-60.895,176.979,15.443,151.897
C09702=1100.062,111.194,-60.876,176.975,15.443,151.897
C09703=1100.056,110.945,-60.857,176.973,15.443,151.898
C09704=1100.050,110.696,-60.838,176.969,15.443,151.899
C09705=1100.045,110.447,-60.819,176.967,15.443,151.899
C09706=1100.039,110.197,-60.801,176.964,15.443,151.900
C09707=1100.033,109.948,-60.782,176.961,15.443,151.900
C09708=1100.028,109.699,-60.763,176.958,15.442,151.901
C09709=1100.021,109.450,-60.744,176.955,15.442,151.901
C09710=1100.016,109.200,-60.725,176.952,15.442,151.902
C09711=1100.011,108.951,-60.707,176.949,15.443,151.903
C09712=1100.004,108.702,-60.688,176.946,15.442,151.903
C09713=1099.999,108.452,-60.669,176.943,15.442,151.904
C09714=1099.994,108.204,-60.650,176.940,15.442,151.905
C09715=1099.987,107.954,-60.632,176.938,15.442,151.905
C09716=1099.982,107.705,-60.613,176.934,15.441,151.906
C09717=1099.976,107.456,-60.595,176.932,15.442,151.906
C09718=1099.971,107.206,-60.576,176.929,15.441,151.907
C09719=1099.966,106.957,-60.557,176.926,15.441,151.907
C09720=1099.959,106.708,-60.539,176.923,15.441,151.908
C09721=1099.954,106.458,-60.520,176.920,15.441,151.909
C09722=1099.948,106.210,-60.502,176.917,15.441,151.909
C09723=1099.942,105.960,-60.483,176.914,15.441,151.910
C09724=1099.937,105.711,-60.464,176.911,15.441,151.910
C09725=1099.931,105.462,-60.446,176.908,15.440,151.911
C09726=1099.925,105.212,-60.427,176.905,15.440,151.912
C09727=1099.920,104.963,-60.409,176.902,15.440,151.912
C09728=1099.914,104.714,-60.390,176.900,15.440,151.913
C09729=1099.909,104.465,-60.372,176.896,15.440,151.913
C09730=1099.903,104.215,-60.353,176.894,15.440,151.914
C09731=1099.897,103.966,-60.334,176.891,15.439,151.915
C09732=1099.892,103.717,-60.316,176.888,15.439,151.915
C09733=1099.886,103.468,-60.297,176.885,15.439,151.916
C09734=1099.880,103.218,-60.279,176.883,15.439,151.916
C09735=1099.875,102.969,-60.260,176.879,15.438,151.917
C09736=1099.869,102.720,-60.243,176.877,15.438,151.917
C09737=1099.864,102.471,-60.223,176.874,15.438,151.918
C09738=1099.858,102.222,-60.206,176.871,15.438,151.918
C09739=1099.852,101.972,-60.186,176.868,15.438,151.919
C09740=1099.847,101.723,-60.169,176.865,15.438,151.920
C09741=1099.841,101.474,-60.150,176.862,15.437,151.920
C09742=1099.836,101.225,-60.132,176.860,15.437,151.921
C09743=1099.830,100.975,-60.113,176.857,15.437,151.921
C09744=1099.824,100.726,-60.095,176.854,15.437,151.922
C09745=1099.818,100.477,-60.077,176.851,15.436,151.922
C09746=1099.813,100.227,-60.058,176.848,15.436,151.923
C09747=1099.807,99.978,-60.041,176.845,15.436,151.923
C09748=1099.801,99.729,-60.022,176.843,15.436,151.924
C09749=1099.796,99.479,-60.004,176.839,15.436,151.925
C09750=1099.789,99.230,-59.985,176.837,15.436,151.925
C09751=1099.784,98.981,-59.968,176.834,15.435,151.926
C09752=1099.779,98.731,-59.949,176.831,15.435,151.926
C09753=1099.773,98.483,-59.931,176.828,15.435,151.927
C09754=1099.767,98.233,-59.913,176.826,15.435,151.927
C09755=1099.762,97.984,-59.895,176.822,15.434,151.928
C09756=1099.755,97.735,-59.876,176.820,15.435,151.929
C09757=1099.750,97.486,-59.858,176.818,15.434,151.929
C09758=1099.745,97.235,-59.840,176.814,15.434,151.930
C09759=1099.739,96.987,-59.822,176.812,15.434,151.930
C09760=1099.733,96.737,-59.804,176.809,15.433,151.931
C09761=1099.728,96.488,-59.785,176.806,15.434,151.931
C09762=1099.721,96.215,-59.766,176.803,15.433,151.932
C09763=1099.715,95.941,-59.746,176.800,15.433,151.932
C09764=1099.708,95.668,-59.726,176.796,15.432,151.933
C09765=1099.703,95.394,-59.706,176.794,15.432,151.934
C09766=1099.697,95.145,-59.688,176.791,15.432,151.934
C09767=1099.691,94.896,-59.670,176.788,15.432,151.935
C09768=1099.686,94.646,-59.652,176.785,15.431,151.935
C09769=1099.680,94.397,-59.634,176.783,15.431,151.936
C09770=1099.674,94.148,-59.616,176.780,15.431,151.936
C09771=1099.668,93.899,-59.598,176.777,15.431,151.937
C09772=1099.663,93.649,-59.579,176.774,15.430,151.937
C09773=1099.657,93.400,-59.562,176.772,15.430,151.938
C09774=1099.651,93.150,-59.544,176.768,15.429,151.938
C09775=1099.646,92.901,-59.526,176.766,15.429,151.939
C09776=1099.641,92.652,-59.508,176.763,15.429,151.939
C09777=1099.635,92.402,-59.490,176.760,15.429,151.940
C09778=1099.629,92.154,-59.472,176.758,15.428,151.940
C09779=1099.624,91.905,-59.454,176.755,15.428,151.941
C09780=1099.617,91.655,-59.436,176.752,15.428,151.942
C09781=1099.613,91.406,-59.418,176.750,15.427,151.942
C09782=1099.607,91.157,-59.401,176.746,15.427,151.943
C09783=1099.601,90.907,-59.383,176.744,15.427,151.943
C09784=1099.596,90.658,-59.365,176.742,15.427,151.943
C09785=1099.589,90.408,-59.347,176.738,15.426,151.944
C09786=1099.584,90.159,-59.330,176.736,15.426,151.944
C09787=1099.578,89.910,-59.312,176.733,15.426,151.945
C09788=1099.572,89.660,-59.294,176.730,15.426,151.946
C09789=1099.567,89.411,-59.277,176.727,15.425,151.946
C09790=1099.561,89.161,-59.259,176.725,15.425,151.947
C09791=1099.555,88.912,-59.241,176.722,15.424,151.947
C09792=1099.550,88.663,-59.224,176.719,15.424,151.948
C09793=1099.543,88.414,-59.206,176.716,15.424,151.948
C09794=1099.538,88.165,-59.188,176.714,15.424,151.949
C09795=1099.532,87.916,-59.171,176.711,15.423,151.949
C09796=1099.526,87.666,-59.153,176.709,15.423,151.950
C09797=1099.521,87.417,-59.135,176.705,15.422,151.950
C09798=1099.515,87.168,-59.118,176.703,15.422,151.951
C09799=1099.509,86.918,-59.100,176.701,15.422,151.951
C09800=1099.504,86.669,-59.082,176.698,15.421,151.952
C09801=1099.498,86.420,-59.064,176.695,15.422,151.952
C09802=1099.492,86.170,-59.047,176.692,15.421,151.953
C09803=1099.486,85.921,-59.029,176.690,15.421,151.953
C09804=1099.481,85.672,-59.011,176.687,15.420,151.954
C09805=1099.475,85.422,-58.993,176.684,15.420,151.954
C09806=1099.470,85.173,-58.977,176.681,15.419,151.955
C09807=1099.464,84.924,-58.959,176.679,15.419,151.955
C09808=1099.459,84.675,-58.941,176.676,15.418,151.956
C09809=1099.452,84.425,-58.924,176.673,15.419,151.956
C09810=1099.447,84.176,-58.906,176.670,15.418,151.957
C09811=1099.441,83.927,-58.888,176.668,15.418,151.957
C09812=1099.436,83.676,-58.871,176.666,15.418,151.958
C09813=1099.430,83.427,-58.854,176.663,15.417,151.958
C09814=1099.425,83.178,-58.836,176.660,15.417,151.959
C09815=1099.419,82.929,-58.818,176.657,15.416,151.959
C09816=1099.413,82.680,-58.801,176.655,15.416,151.960
C09817=1099.408,82.430,-58.784,176.652,15.415,151.960
C09818=1099.402,82.181,-58.766,176.650,15.415,151.961
C09819=1099.396,81.932,-58.749,176.646,15.415,151.961
C09820=1099.390,81.683,-58.732,176.644,15.414,151.962
C09821=1099.385,81.433,-58.714,176.641,15.413,151.962
C09822=1099.379,81.184,-58.697,176.639,15.414,151.963
C09823=1099.374,80.935,-58.679,176.637,15.413,151.963
C09824=1099.368,80.685,-58.662,176.634,15.412,151.963
C09825=1099.363,80.436,-58.645,176.631,15.413,151.964
C09826=1099.356,80.162,-58.626,176.628,15.412,151.964
C09827=1099.350,79.889,-58.607,176.625,15.411,151.965
C09828=1099.344,79.616,-58.588,176.623,15.411,151.965
C09829=1099.337,79.342,-58.568,176.619,15.410,151.966
C09830=1099.332,79.092,-58.552,176.616,15.410,151.966
C09831=1099.327,78.843,-58.534,176.614,15.409,151.967
C09832=1099.321,78.594,-58.517,176.612,15.409,151.967
C09833=1099.315,78.345,-58.500,176.609,15.409,151.968
C09834=1099.309,78.095,-58.482,176.607,15.408,151.968
C09835=1099.304,77.845,-58.465,176.603,15.408,151.969
C09836=1099.298,77.596,-58.448,176.601,15.408,151.969
C09837=1099.292,77.347,-58.432,176.598,15.407,151.970
C09838=1099.287,77.098,-58.414,176.596,15.406,151.970
C09839=1099.281,76.848,-58.396,176.593,15.407,151.971
C09840=1099.275,76.599,-58.379,176.591,15.406,151.971
C09841=1099.269,76.350,-58.362,176.588,15.405,151.972
C09842=1099.264,76.100,-58.345,176.585,15.404,151.972
C09843=1099.258,75.851,-58.328,176.583,15.405,151.973
C09844=1099.252,75.602,-58.312,176.580,15.404,151.973
C09845=1099.246,75.352,-58.294,176.578,15.403,151.973
C09846=1099.241,75.102,-58.277,176.575,15.403,151.974
C09847=1099.235,74.854,-58.260,176.572,15.403,151.974
C09848=1099.230,74.604,-58.243,176.570,15.402,151.975
C09849=1099.224,74.355,-58.225,176.567,15.402,151.975
C09850=1099.218,74.106,-58.209,176.565,15.401,151.976
C09851=1099.213,73.857,-58.192,176.562,15.400,151.976
C09852=1099.207,73.607,-58.175,176.559,15.401,151.977
C09853=1099.201,73.357,-58.157,176.557,15.400,151.977
C09854=1099.195,73.108,-58.141,176.554,15.399,151.977
C09855=1099.190,72.858,-58.124,176.552,15.399,151.978
C09856=1099.184,72.609,-58.107,176.549,15.398,151.978
C09857=1099.179,72.360,-58.090,176.547,15.398,151.979
C09858=1099.172,72.111,-58.073,176.544,15.397,151.979
C09859=1099.167,71.861,-58.056,176.542,15.397,151.980
C09860=1099.162,71.612,-58.039,176.539,15.396,151.980
C09861=1099.156,71.363,-58.022,176.536,15.396,151.981
C09862=1099.151,71.113,-58.005,176.534,15.396,151.981
C09863=1099.145,70.864,-57.989,176.531,15.395,151.981
C09864=1099.139,70.615,-57.972,176.529,15.395,151.982
C09865=1099.133,70.365,-57.954,176.526,15.394,151.982
C09866=1099.127,70.115,-57.938,176.524,15.393,151.983
C09867=1099.122,69.866,-57.921,176.521,15.392,151.983
C09868=1099.116,69.617,-57.904,176.519,15.392,151.984
C09869=1099.111,69.367,-57.887,176.516,15.392,151.984
C09870=1099.104,69.118,-57.870,176.513,15.391,151.985
C09871=1099.099,68.869,-57.854,176.511,15.391,151.985
C09872=1099.093,68.619,-57.837,176.508,15.390,151.985
C09873=1099.088,68.370,-57.820,176.506,15.390,151.986
C09874=1099.082,68.121,-57.803,176.504,15.390,151.986
C09875=1099.077,67.871,-57.787,176.501,15.389,151.987
C09876=1099.071,67.622,-57.770,176.499,15.389,151.987
C09877=1099.065,67.372,-57.754,176.496,15.388,151.988
C09878=1099.059,67.124,-57.737,176.493,15.387,151.988
C09879=1099.054,66.874,-57.720,176.491,15.387,151.988
C09880=1099.048,66.625,-57.703,176.488,15.386,151.989
C09881=1099.042,66.375,-57.687,176.486,15.386,151.989
C09882=1099.037,66.126,-57.670,176.483,15.385,151.990
C09883=1099.031,65.876,-57.654,176.481,15.385,151.990
C09884=1099.025,65.627,-57.637,176.478,15.384,151.990
C09885=1099.019,65.378,-57.620,176.476,15.384,151.991
C09886=1099.013,65.129,-57.604,176.474,15.383,151.991
C09887=1099.008,64.879,-57.587,176.471,15.382,151.992
C09888=1099.002,64.630,-57.571,176.468,15.382,151.992
C09889=1098.997,64.380,-57.554,176.465,15.381,151.993
C09890=1098.990,64.107,-57.536,176.463,15.381,151.993
C09891=1098.984,63.833,-57.517,176.460,15.380,151.993
C09892=1098.977,63.559,-57.500,176.458,15.380,151.994
C09893=1098.971,63.286,-57.482,176.455,15.379,151.994
C09894=1098.966,63.036,-57.465,176.453,15.379,151.995
C09895=1098.959,62.787,-57.448,176.450,15.378,151.995
C09896=1098.953,62.538,-57.432,176.448,15.378,151.996
C09897=1098.947,62.289,-57.416,176.445,15.377,151.996
C09898=1098.942,62.039,-57.399,176.442,15.377,151.997
C09899=1098.936,61.790,-57.383,176.440,15.377,151.997
C09900=1098.930,61.540,-57.366,176.437,15.376,151.997
C09901=1098.924,61.291,-57.350,176.435,15.375,151.998
C09902=1098.918,61.041,-57.334,176.432,15.374,151.998
C09903=1098.913,60.792,-57.317,176.430,15.374,151.999
C09904=1098.907,60.542,-57.301,176.428,15.374,151.999
C09905=1098.901,60.293,-57.284,176.425,15.373,151.999
C09906=1098.895,60.044,-57.268,176.423,15.372,152.000
C09907=1098.889,59.794,-57.252,176.421,15.372,152.000
C09908=1098.884,59.545,-57.235,176.418,15.371,152.001
C09909=1098.878,59.295,-57.219,176.415,15.371,152.001
C09910=1098.872,59.046,-57.203,176.413,15.370,152.001
C09911=1098.867,58.797,-57.187,176.410,15.370,152.002
C09912=1098.861,58.547,-57.171,176.408,15.369,152.002
C09913=1098.855,58.298,-57.155,176.405,15.369,152.003
C09914=1098.850,58.048,-57.138,176.403,15.368,152.003
C09915=1098.844,57.799,-57.122,176.400,15.367,152.003
C09916=1098.838,57.550,-57.105,176.398,15.367,152.004
C09917=1098.832,57.300,-57.089,176.396,15.366,152.004
C09918=1098.826,57.051,-57.073,176.393,15.365,152.005
C09919=1098.820,56.802,-57.057,176.391,15.365,152.005
C09920=1098.815,56.551,-57.041,176.389,15.364,152.005
C09921=1098.810,56.302,-57.024,176.386,15.364,152.006
C09922=1098.804,56.053,-57.008,176.384,15.363,152.006
C09923=1098.798,55.804,-56.992,176.381,15.362,152.007
C09924=1098.792,55.555,-56.976,176.379,15.362,152.007
C09925=1098.786,55.305,-56.960,176.377,15.361,152.007
C09926=1098.781,55.055,-56.944,176.374,15.360,152.008
C09927=1098.775,54.806,-56.928,176.372,15.360,152.008
C09928=1098.770,54.556,-56.911,176.369,15.360,152.009
C09929=1098.764,54.308,-56.895,176.367,15.359,152.009
C09930=1098.759,54.058,-56.880,176.365,15.358,152.009
C09931=1098.753,53.808,-56.863,176.362,15.357,152.010
C09932=1098.747,53.559,-56.847,176.359,15.357,152.010
C09933=1098.741,53.310,-56.831,176.358,15.356,152.010
C09934=1098.735,53.060,-56.815,176.355,15.356,152.011
C09935=1098.730,52.811,-56.799,176.352,15.355,152.011
C09936=1098.724,52.562,-56.783,176.350,15.355,152.011
C09937=1098.718,52.312,-56.767,176.348,15.354,152.012
C09938=1098.712,52.062,-56.751,176.345,15.353,152.012
C09939=1098.706,51.813,-56.735,176.342,15.352,152.013
C09940=1098.702,51.564,-56.719,176.340,15.352,152.013
C09941=1098.696,51.314,-56.703,176.338,15.351,152.013
C09942=1098.690,51.065,-56.687,176.335,15.351,152.014
C09943=1098.684,50.816,-56.671,176.333,15.350,152.014
C09944=1098.678,50.566,-56.655,176.331,15.350,152.015
C09945=1098.673,50.317,-56.639,176.329,15.348,152.015
C09946=1098.667,50.067,-56.624,176.326,15.348,152.015
C09947=1098.661,49.818,-56.607,176.324,15.348,152.016
C09948=1098.655,49.568,-56.591,176.322,15.346,152.016
C09949=1098.650,49.319,-56.576,176.319,15.346,152.016
C09950=1098.644,49.070,-56.560,176.316,15.345,152.017
C09951=1098.639,48.820,-56.544,176.315,15.344,152.017
C09952=1098.633,48.571,-56.528,176.312,15.344,152.017
C09953=1098.628,48.321,-56.513,176.310,15.343,152.018
C09954=1098.621,48.048,-56.495,176.307,15.343,152.018
C09955=1098.615,47.774,-56.477,176.305,15.342,152.019
C09956=1098.609,47.500,-56.460,176.302,15.341,152.019
C09957=1098.603,47.226,-56.442,176.300,15.340,152.019
C09958=1098.597,46.976,-56.427,176.297,15.340,152.020
C09959=1098.592,46.728,-56.411,176.295,15.338,152.020
C09960=1098.586,46.478,-56.395,176.293,15.338,152.020
C09961=1098.580,46.228,-56.379,176.291,15.337,152.021
C09962=1098.575,45.979,-56.364,176.288,15.337,152.021
C09963=1098.570,45.729,-56.348,176.286,15.336,152.021
C09964=1098.564,45.480,-56.332,176.284,15.335,152.022
C09965=1098.558,45.231,-56.318,176.281,15.334,152.022
C09966=1098.552,44.981,-56.301,176.279,15.334,152.022
C09967=1098.546,44.731,-56.286,176.276,15.333,152.023
C09968=1098.541,44.483,-56.270,176.274,15.332,152.023
C09969=1098.535,44.233,-56.254,176.272,15.332,152.023
C09970=1098.530,43.983,-56.239,176.269,15.331,152.024
C09971=1098.524,43.734,-56.223,176.267,15.330,152.024
C09972=1098.519,43.484,-56.207,176.265,15.330,152.025
C09973=1098.513,43.235,-56.191,176.262,15.328,152.025
C09974=1098.508,42.986,-56.176,176.260,15.328,152.025
C09975=1098.501,42.736,-56.161,176.258,15.327,152.025
C09976=1098.495,42.487,-56.145,176.255,15.326,152.026
C09977=1098.490,42.237,-56.130,176.253,15.326,152.026
C09978=1098.485,41.987,-56.114,176.251,15.325,152.027
C09979=1098.478,41.738,-56.098,176.248,15.325,152.027
C09980=1098.473,41.489,-56.083,176.247,15.324,152.027
C09981=1098.467,41.239,-56.068,176.245,15.323,152.028
C09982=1098.461,40.990,-56.051,176.242,15.322,152.028
C09983=1098.456,40.740,-56.036,176.240,15.321,152.028
C09984=1098.450,40.491,-56.021,176.238,15.321,152.029
C09985=1098.444,40.241,-56.005,176.235,15.320,152.029
C09986=1098.439,39.992,-55.990,176.233,15.320,152.029
C09987=1098.433,39.742,-55.974,176.231,15.319,152.030
C09988=1098.427,39.493,-55.960,176.228,15.318,152.030
C09989=1098.421,39.244,-55.943,176.226,15.317,152.030
C09990=1098.416,38.994,-55.928,176.224,15.317,152.031
C09991=1098.410,38.745,-55.913,176.221,15.316,152.031
C09992=1098.404,38.495,-55.898,176.219,15.315,152.031
C09993=1098.399,38.246,-55.882,176.217,15.315,152.032
C09994=1098.393,37.996,-55.866,176.214,15.313,152.032
C09995=1098.387,37.747,-55.851,176.212,15.313,152.032
C09996=1098.382,37.498,-55.836,176.210,15.312,152.033
//INST
///DATE 2021/06/17 10:53
///ATTR SC,RW,RJ
////FRAME ROBOT
///GROUP1 RB1
NOP
MOVL C00000 V=800.0 PL=0
MOVL C00001 V=800.0 PL=0
MOVL C00002 V=800.0 PL=0
MOVL C00003 V=800.0 PL=0
MOVL C00004 V=800.0 PL=0
MOVL C00005 V=800.0 PL=0
MOVL C00006 V=800.0 PL=0
MOVL C00007 V=800.0 PL=0
MOVL C00008 V=800.0 PL=0
MOVL C00009 V=800.0 PL=0
MOVL C00010 V=800.0 PL=0
MOVL C00011 V=800.0 PL=0
MOVL C00012 V=800.0 PL=0
MOVL C00013 V=800.0 PL=0
MOVL C00014 V=800.0 PL=0
MOVL C00015 V=800.0 PL=0
MOVL C00016 V=800.0 PL=0
MOVL C00017 V=800.0 PL=0
MOVL C00018 V=800.0 PL=0
MOVL C00019 V=800.0 PL=0
MOVL C00020 V=800.0 PL=0
MOVL C00021 V=800.0 PL=0
MOVL C00022 V=800.0 PL=0
MOVL C00023 V=800.0 PL=0
MOVL C00024 V=800.0 PL=0
MOVL C00025 V=800.0 PL=0
MOVL C00026 V=800.0 PL=0
MOVL C00027 V=800.0 PL=0
MOVL C00028 V=800.0 PL=0
MOVL C00029 V=800.0 PL=0
MOVL C00030 V=800.0 PL=0
MOVL C00031 V=800.0 PL=0
MOVL C00032 V=800.0 PL=0
MOVL C00033 V=800.0 PL=0
MOVL C00034 V=800.0 PL=0
MOVL C00035 V=800.0 PL=0
MOVL C00036 V=800.0 PL=0
MOVL C00037 V=800.0 PL=0
MOVL C00038 V=800.0 PL=0
MOVL C00039 V=800.0 PL=0
MOVL C00040 V=800.0 PL=0
MOVL C00041 V=800.0 PL=0
MOVL C00042 V=800.0 PL=0
MOVL C00043 V=800.0 PL=0
MOVL C00044 V=800.0 PL=0
MOVL C00045 V=800.0 PL=0
MOVL C00046 V=800.0 PL=0
MOVL C00047 V=800.0 PL=0
MOVL C00048 V=800.0 PL=0
MOVL C00049 V=800.0 PL=0
MOVL C00050 V=800.0 PL=0
MOVL C00051 V=800.0 PL=0
MOVL C00052 V=800.0 PL=0
MOVL C00053 V=800.0 PL=0
MOVL C00054 V=800.0 PL=0
MOVL C00055 V=800.0 PL=0
MOVL C00056 V=800.0 PL=0
MOVL C00057 V=800.0 PL=0
MOVL C00058 V=800.0 PL=0
MOVL C00059 V=800.0 PL=0
MOVL C00060 V=800.0 PL=0
MOVL C00061 V=800.0 PL=0
MOVL C00062 V=800.0 PL=0
MOVL C00063 V=800.0 PL=0
MOVL C00064 V=800.0 PL=0
MOVL C00065 V=800.0 PL=0
MOVL C00066 V=800.0 PL=0
MOVL C00067 V=800.0 PL=0
MOVL C00068 V=800.0 PL=0
MOVL C00069 V=800.0 PL=0
MOVL C00070 V=800.0 PL=0
MOVL C00071 V=800.0 PL=0
MOVL C00072 V=800.0 PL=0
MOVL C00073 V=800.0 PL=0
MOVL C00074 V=800.0 PL=0
MOVL C00075 V=800.0 PL=0
MOVL C00076 V=800.0 PL=0
MOVL C00077 V=800.0 PL=0
MOVL C00078 V=800.0 PL=0
MOVL C00079 V=800.0 PL=0
MOVL C00080 V=800.0 PL=0
MOVL C00081 V=800.0 PL=0
MOVL C00082 V=800.0 PL=0
MOVL C00083 V=800.0 PL=0
MOVL C00084 V=800.0 PL=0
MOVL C00085 V=800.0 PL=0
MOVL C00086 V=800.0 PL=0
MOVL C00087 V=800.0 PL=0
MOVL C00088 V=800.0 PL=0
MOVL C00089 V=800.0 PL=0
MOVL C00090 V=800.0 PL=0
MOVL C00091 V=800.0 PL=0
MOVL C00092 V=800.0 PL=0
MOVL C00093 V=800.0 PL=0
MOVL C00094 V=800.0 PL=0
MOVL C00095 V=800.0 PL=0
MOVL C00096 V=800.0 PL=0
MOVL C00097 V=800.0 PL=0
MOVL C00098 V=800.0 PL=0
MOVL C00099 V=800.0 PL=0
MOVL C00100 V=800.0 PL=0
MOVL C00101 V=800.0 PL=0
MOVL C00102 V=800.0 PL=0
MOVL C00103 V=800.0 PL=0
MOVL C00104 V=800.0 PL=0
MOVL C00105 V=800.0 PL=0
MOVL C00106 V=800.0 PL=0
MOVL C00107 V=800.0 PL=0
MOVL C00108 V=800.0 PL=0
MOVL C00109 V=800.0 PL=0
MOVL C00110 V=800.0 PL=0
MOVL C00111 V=800.0 PL=0
MOVL C00112 V=800.0 PL=0
MOVL C00113 V=800.0 PL=0
MOVL C00114 V=800.0 PL=0
MOVL C00115 V=800.0 PL=0
MOVL C00116 V=800.0 PL=0
MOVL C00117 V=800.0 PL=0
MOVL C00118 V=800.0 PL=0
MOVL C00119 V=800.0 PL=0
MOVL C00120 V=800.0 PL=0
MOVL C00121 V=800.0 PL=0
MOVL C00122 V=800.0 PL=0
MOVL C00123 V=800.0 PL=0
MOVL C00124 V=800.0 PL=0
MOVL C00125 V=800.0 PL=0
MOVL C00126 V=800.0 PL=0
MOVL C00127 V=800.0 PL=0
MOVL C00128 V=800.0 PL=0
MOVL C00129 V=800.0 PL=0
MOVL C00130 V=800.0 PL=0
MOVL C00131 V=800.0 PL=0
MOVL C00132 V=800.0 PL=0
MOVL C00133 V=800.0 PL=0
MOVL C00134 V=800.0 PL=0
MOVL C00135 V=800.0 PL=0
MOVL C00136 V=800.0 PL=0
MOVL C00137 V=800.0 PL=0
MOVL C00138 V=800.0 PL=0
MOVL C00139 V=800.0 PL=0
MOVL C00140 V=800.0 PL=0
MOVL C00141 V=800.0 PL=0
MOVL C00142 V=800.0 PL=0
MOVL C00143 V=800.0 PL=0
MOVL C00144 V=800.0 PL=0
MOVL C00145 V=800.0 PL=0
MOVL C00146 V=800.0 PL=0
MOVL C00147 V=800.0 PL=0
MOVL C00148 V=800.0 PL=0
MOVL C00149 V=800.0 PL=0
MOVL C00150 V=800.0 PL=0
MOVL C00151 V=800.0 PL=0
MOVL C00152 V=800.0 PL=0
MOVL C00153 V=800.0 PL=0
MOVL C00154 V=800.0 PL=0
MOVL C00155 V=800.0 PL=0
MOVL C00156 V=800.0 PL=0
MOVL C00157 V=800.0 PL=0
MOVL C00158 V=800.0 PL=0
MOVL C00159 V=800.0 PL=0
MOVL C00160 V=800.0 PL=0
MOVL C00161 V=800.0 PL=0
MOVL C00162 V=800.0 PL=0
MOVL C00163 V=800.0 PL=0
MOVL C00164 V=800.0 PL=0
MOVL C00165 V=800.0 PL=0
MOVL C00166 V=800.0 PL=0
MOVL C00167 V=800.0 PL=0
MOVL C00168 V=800.0 PL=0
MOVL C00169 V=800.0 PL=0
MOVL C00170 V=800.0 PL=0
MOVL C00171 V=800.0 PL=0
MOVL C00172 V=800.0 PL=0
MOVL C00173 V=800.0 PL=0
MOVL C00174 V=800.0 PL=0
MOVL C00175 V=800.0 PL=0
MOVL C00176 V=800.0 PL=0
MOVL C00177 V=800.0 PL=0
MOVL C00178 V=800.0 PL=0
MOVL C00179 V=800.0 PL=0
MOVL C00180 V=800.0 PL=0
MOVL C00181 V=800.0 PL=0
MOVL C00182 V=800.0 PL=0
MOVL C00183 V=800.0 PL=0
MOVL C00184 V=800.0 PL=0
MOVL C00185 V=800.0 PL=0
MOVL C00186 V=800.0 PL=0
MOVL C00187 V=800.0 PL=0
MOVL C00188 V=800.0 PL=0
MOVL C00189 V=800.0 PL=0
MOVL C00190 V=800.0 PL=0
MOVL C00191 V=800.0 PL=0
MOVL C00192 V=800.0 PL=0
MOVL C00193 V=800.0 PL=0
MOVL C00194 V=800.0 PL=0
MOVL C00195 V=800.0 PL=0
MOVL C00196 V=800.0 PL=0
MOVL C00197 V=800.0 PL=0
MOVL C00198 V=800.0 PL=0
MOVL C00199 V=800.0 PL=0
MOVL C00200 V=800.0 PL=0
MOVL C00201 V=800.0 PL=0
MOVL C00202 V=800.0 PL=0
MOVL C00203 V=800.0 PL=0
MOVL C00204 V=800.0 PL=0
MOVL C00205 V=800.0 PL=0
MOVL C00206 V=800.0 PL=0
MOVL C00207 V=800.0 PL=0
MOVL C00208 V=800.0 PL=0
MOVL C00209 V=800.0 PL=0
MOVL C00210 V=800.0 PL=0
MOVL C00211 V=800.0 PL=0
MOVL C00212 V=800.0 PL=0
MOVL C00213 V=800.0 PL=0
MOVL C00214 V=800.0 PL=0
MOVL C00215 V=800.0 PL=0
MOVL C00216 V=800.0 PL=0
MOVL C00217 V=800.0 PL=0
MOVL C00218 V=800.0 PL=0
MOVL C00219 V=800.0 PL=0
MOVL C00220 V=800.0 PL=0
MOVL C00221 V=800.0 PL=0
MOVL C00222 V=800.0 PL=0
MOVL C00223 V=800.0 PL=0
MOVL C00224 V=800.0 PL=0
MOVL C00225 V=800.0 PL=0
MOVL C00226 V=800.0 PL=0
MOVL C00227 V=800.0 PL=0
MOVL C00228 V=800.0 PL=0
MOVL C00229 V=800.0 PL=0
MOVL C00230 V=800.0 PL=0
MOVL C00231 V=800.0 PL=0
MOVL C00232 V=800.0 PL=0
MOVL C00233 V=800.0 PL=0
MOVL C00234 V=800.0 PL=0
MOVL C00235 V=800.0 PL=0
MOVL C00236 V=800.0 PL=0
MOVL C00237 V=800.0 PL=0
MOVL C00238 V=800.0 PL=0
MOVL C00239 V=800.0 PL=0
MOVL C00240 V=800.0 PL=0
MOVL C00241 V=800.0 PL=0
MOVL C00242 V=800.0 PL=0
MOVL C00243 V=800.0 PL=0
MOVL C00244 V=800.0 PL=0
MOVL C00245 V=800.0 PL=0
MOVL C00246 V=800.0 PL=0
MOVL C00247 V=800.0 PL=0
MOVL C00248 V=800.0 PL=0
MOVL C00249 V=800.0 PL=0
MOVL C00250 V=800.0 PL=0
MOVL C00251 V=800.0 PL=0
MOVL C00252 V=800.0 PL=0
MOVL C00253 V=800.0 PL=0
MOVL C00254 V=800.0 PL=0
MOVL C00255 V=800.0 PL=0
MOVL C00256 V=800.0 PL=0
MOVL C00257 V=800.0 PL=0
MOVL C00258 V=800.0 PL=0
MOVL C00259 V=800.0 PL=0
MOVL C00260 V=800.0 PL=0
MOVL C00261 V=800.0 PL=0
MOVL C00262 V=800.0 PL=0
MOVL C00263 V=800.0 PL=0
MOVL C00264 V=800.0 PL=0
MOVL C00265 V=800.0 PL=0
MOVL C00266 V=800.0 PL=0
MOVL C00267 V=800.0 PL=0
MOVL C00268 V=800.0 PL=0
MOVL C00269 V=800.0 PL=0
MOVL C00270 V=800.0 PL=0
MOVL C00271 V=800.0 PL=0
MOVL C00272 V=800.0 PL=0
MOVL C00273 V=800.0 PL=0
MOVL C00274 V=800.0 PL=0
MOVL C00275 V=800.0 PL=0
MOVL C00276 V=800.0 PL=0
MOVL C00277 V=800.0 PL=0
MOVL C00278 V=800.0 PL=0
MOVL C00279 V=800.0 PL=0
MOVL C00280 V=800.0 PL=0
MOVL C00281 V=800.0 PL=0
MOVL C00282 V=800.0 PL=0
MOVL C00283 V=800.0 PL=0
MOVL C00284 V=800.0 PL=0
MOVL C00285 V=800.0 PL=0
MOVL C00286 V=800.0 PL=0
MOVL C00287 V=800.0 PL=0
MOVL C00288 V=800.0 PL=0
MOVL C00289 V=800.0 PL=0
MOVL C00290 V=800.0 PL=0
MOVL C00291 V=800.0 PL=0
MOVL C00292 V=800.0 PL=0
MOVL C00293 V=800.0 PL=0
MOVL C00294 V=800.0 PL=0
MOVL C00295 V=800.0 PL=0
MOVL C00296 V=800.0 PL=0
MOVL C00297 V=800.0 PL=0
MOVL C00298 V=800.0 PL=0
MOVL C00299 V=800.0 PL=0
MOVL C00300 V=800.0 PL=0
MOVL C00301 V=800.0 PL=0
MOVL C00302 V=800.0 PL=0
MOVL C00303 V=800.0 PL=0
MOVL C00304 V=800.0 PL=0
MOVL C00305 V=800.0 PL=0
MOVL C00306 V=800.0 PL=0
MOVL C00307 V=800.0 PL=0
MOVL C00308 V=800.0 PL=0
MOVL C00309 V=800.0 PL=0
MOVL C00310 V=800.0 PL=0
MOVL C00311 V=800.0 PL=0
MOVL C00312 V=800.0 PL=0
MOVL C00313 V=800.0 PL=0
MOVL C00314 V=800.0 PL=0
MOVL C00315 V=800.0 PL=0
MOVL C00316 V=800.0 PL=0
MOVL C00317 V=800.0 PL=0
MOVL C00318 V=800.0 PL=0
MOVL C00319 V=800.0 PL=0
MOVL C00320 V=800.0 PL=0
MOVL C00321 V=800.0 PL=0
MOVL C00322 V=800.0 PL=0
MOVL C00323 V=800.0 PL=0
MOVL C00324 V=800.0 PL=0
MOVL C00325 V=800.0 PL=0
MOVL C00326 V=800.0 PL=0
MOVL C00327 V=800.0 PL=0
MOVL C00328 V=800.0 PL=0
MOVL C00329 V=800.0 PL=0
MOVL C00330 V=800.0 PL=0
MOVL C00331 V=800.0 PL=0
MOVL C00332 V=800.0 PL=0
MOVL C00333 V=800.0 PL=0
MOVL C00334 V=800.0 PL=0
MOVL C00335 V=800.0 PL=0
MOVL C00336 V=800.0 PL=0
MOVL C00337 V=800.0 PL=0
MOVL C00338 V=800.0 PL=0
MOVL C00339 V=800.0 PL=0
MOVL C00340 V=800.0 PL=0
MOVL C00341 V=800.0 PL=0
MOVL C00342 V=800.0 PL=0
MOVL C00343 V=800.0 PL=0
MOVL C00344 V=800.0 PL=0
MOVL C00345 V=800.0 PL=0
MOVL C00346 V=800.0 PL=0
MOVL C00347 V=800.0 PL=0
MOVL C00348 V=800.0 PL=0
MOVL C00349 V=800.0 PL=0
MOVL C00350 V=800.0 PL=0
MOVL C00351 V=800.0 PL=0
MOVL C00352 V=800.0 PL=0
MOVL C00353 V=800.0 PL=0
MOVL C00354 V=800.0 PL=0
MOVL C00355 V=800.0 PL=0
MOVL C00356 V=800.0 PL=0
MOVL C00357 V=800.0 PL=0
MOVL C00358 V=800.0 PL=0
MOVL C00359 V=800.0 PL=0
MOVL C00360 V=800.0 PL=0
MOVL C00361 V=800.0 PL=0
MOVL C00362 V=800.0 PL=0
MOVL C00363 V=800.0 PL=0
MOVL C00364 V=800.0 PL=0
MOVL C00365 V=800.0 PL=0
MOVL C00366 V=800.0 PL=0
MOVL C00367 V=800.0 PL=0
MOVL C00368 V=800.0 PL=0
MOVL C00369 V=800.0 PL=0
MOVL C00370 V=800.0 PL=0
MOVL C00371 V=800.0 PL=0
MOVL C00372 V=800.0 PL=0
MOVL C00373 V=800.0 PL=0
MOVL C00374 V=800.0 PL=0
MOVL C00375 V=800.0 PL=0
MOVL C00376 V=800.0 PL=0
MOVL C00377 V=800.0 PL=0
MOVL C00378 V=800.0 PL=0
MOVL C00379 V=800.0 PL=0
MOVL C00380 V=800.0 PL=0
MOVL C00381 V=800.0 PL=0
MOVL C00382 V=800.0 PL=0
MOVL C00383 V=800.0 PL=0
MOVL C00384 V=800.0 PL=0
MOVL C00385 V=800.0 PL=0
MOVL C00386 V=800.0 PL=0
MOVL C00387 V=800.0 PL=0
MOVL C00388 V=800.0 PL=0
MOVL C00389 V=800.0 PL=0
MOVL C00390 V=800.0 PL=0
MOVL C00391 V=800.0 PL=0
MOVL C00392 V=800.0 PL=0
MOVL C00393 V=800.0 PL=0
MOVL C00394 V=800.0 PL=0
MOVL C00395 V=800.0 PL=0
MOVL C00396 V=800.0 PL=0
MOVL C00397 V=800.0 PL=0
MOVL C00398 V=800.0 PL=0
MOVL C00399 V=800.0 PL=0
MOVL C00400 V=800.0 PL=0
MOVL C00401 V=800.0 PL=0
MOVL C00402 V=800.0 PL=0
MOVL C00403 V=800.0 PL=0
MOVL C00404 V=800.0 PL=0
MOVL C00405 V=800.0 PL=0
MOVL C00406 V=800.0 PL=0
MOVL C00407 V=800.0 PL=0
MOVL C00408 V=800.0 PL=0
MOVL C00409 V=800.0 PL=0
MOVL C00410 V=800.0 PL=0
MOVL C00411 V=800.0 PL=0
MOVL C00412 V=800.0 PL=0
MOVL C00413 V=800.0 PL=0
MOVL C00414 V=800.0 PL=0
MOVL C00415 V=800.0 PL=0
MOVL C00416 V=800.0 PL=0
MOVL C00417 V=800.0 PL=0
MOVL C00418 V=800.0 PL=0
MOVL C00419 V=800.0 PL=0
MOVL C00420 V=800.0 PL=0
MOVL C00421 V=800.0 PL=0
MOVL C00422 V=800.0 PL=0
MOVL C00423 V=800.0 PL=0
MOVL C00424 V=800.0 PL=0
MOVL C00425 V=800.0 PL=0
MOVL C00426 V=800.0 PL=0
MOVL C00427 V=800.0 PL=0
MOVL C00428 V=800.0 PL=0
MOVL C00429 V=800.0 PL=0
MOVL C00430 V=800.0 PL=0
MOVL C00431 V=800.0 PL=0
MOVL C00432 V=800.0 PL=0
MOVL C00433 V=800.0 PL=0
MOVL C00434 V=800.0 PL=0
MOVL C00435 V=800.0 PL=0
MOVL C00436 V=800.0 PL=0
MOVL C00437 V=800.0 PL=0
MOVL C00438 V=800.0 PL=0
MOVL C00439 V=800.0 PL=0
MOVL C00440 V=800.0 PL=0
MOVL C00441 V=800.0 PL=0
MOVL C00442 V=800.0 PL=0
MOVL C00443 V=800.0 PL=0
MOVL C00444 V=800.0 PL=0
MOVL C00445 V=800.0 PL=0
MOVL C00446 V=800.0 PL=0
MOVL C00447 V=800.0 PL=0
MOVL C00448 V=800.0 PL=0
MOVL C00449 V=800.0 PL=0
MOVL C00450 V=800.0 PL=0
MOVL C00451 V=800.0 PL=0
MOVL C00452 V=800.0 PL=0
MOVL C00453 V=800.0 PL=0
MOVL C00454 V=800.0 PL=0
MOVL C00455 V=800.0 PL=0
MOVL C00456 V=800.0 PL=0
MOVL C00457 V=800.0 PL=0
MOVL C00458 V=800.0 PL=0
MOVL C00459 V=800.0 PL=0
MOVL C00460 V=800.0 PL=0
MOVL C00461 V=800.0 PL=0
MOVL C00462 V=800.0 PL=0
MOVL C00463 V=800.0 PL=0
MOVL C00464 V=800.0 PL=0
MOVL C00465 V=800.0 PL=0
MOVL C00466 V=800.0 PL=0
MOVL C00467 V=800.0 PL=0
MOVL C00468 V=800.0 PL=0
MOVL C00469 V=800.0 PL=0
MOVL C00470 V=800.0 PL=0
MOVL C00471 V=800.0 PL=0
MOVL C00472 V=800.0 PL=0
MOVL C00473 V=800.0 PL=0
MOVL C00474 V=800.0 PL=0
MOVL C00475 V=800.0 PL=0
MOVL C00476 V=800.0 PL=0
MOVL C00477 V=800.0 PL=0
MOVL C00478 V=800.0 PL=0
MOVL C00479 V=800.0 PL=0
MOVL C00480 V=800.0 PL=0
MOVL C00481 V=800.0 PL=0
MOVL C00482 V=800.0 PL=0
MOVL C00483 V=800.0 PL=0
MOVL C00484 V=800.0 PL=0
MOVL C00485 V=800.0 PL=0
MOVL C00486 V=800.0 PL=0
MOVL C00487 V=800.0 PL=0
MOVL C00488 V=800.0 PL=0
MOVL C00489 V=800.0 PL=0
MOVL C00490 V=800.0 PL=0
MOVL C00491 V=800.0 PL=0
MOVL C00492 V=800.0 PL=0
MOVL C00493 V=800.0 PL=0
MOVL C00494 V=800.0 PL=0
MOVL C00495 V=800.0 PL=0
MOVL C00496 V=800.0 PL=0
MOVL C00497 V=800.0 PL=0
MOVL C00498 V=800.0 PL=0
MOVL C00499 V=800.0 PL=0
MOVL C00500 V=800.0 PL=0
MOVL C00501 V=800.0 PL=0
MOVL C00502 V=800.0 PL=0
MOVL C00503 V=800.0 PL=0
MOVL C00504 V=800.0 PL=0
MOVL C00505 V=800.0 PL=0
MOVL C00506 V=800.0 PL=0
MOVL C00507 V=800.0 PL=0
MOVL C00508 V=800.0 PL=0
MOVL C00509 V=800.0 PL=0
MOVL C00510 V=800.0 PL=0
MOVL C00511 V=800.0 PL=0
MOVL C00512 V=800.0 PL=0
MOVL C00513 V=800.0 PL=0
MOVL C00514 V=800.0 PL=0
MOVL C00515 V=800.0 PL=0
MOVL C00516 V=800.0 PL=0
MOVL C00517 V=800.0 PL=0
MOVL C00518 V=800.0 PL=0
MOVL C00519 V=800.0 PL=0
MOVL C00520 V=800.0 PL=0
MOVL C00521 V=800.0 PL=0
MOVL C00522 V=800.0 PL=0
MOVL C00523 V=800.0 PL=0
MOVL C00524 V=800.0 PL=0
MOVL C00525 V=800.0 PL=0
MOVL C00526 V=800.0 PL=0
MOVL C00527 V=800.0 PL=0
MOVL C00528 V=800.0 PL=0
MOVL C00529 V=800.0 PL=0
MOVL C00530 V=800.0 PL=0
MOVL C00531 V=800.0 PL=0
MOVL C00532 V=800.0 PL=0
MOVL C00533 V=800.0 PL=0
MOVL C00534 V=800.0 PL=0
MOVL C00535 V=800.0 PL=0
MOVL C00536 V=800.0 PL=0
MOVL C00537 V=800.0 PL=0
MOVL C00538 V=800.0 PL=0
MOVL C00539 V=800.0 PL=0
MOVL C00540 V=800.0 PL=0
MOVL C00541 V=800.0 PL=0
MOVL C00542 V=800.0 PL=0
MOVL C00543 V=800.0 PL=0
MOVL C00544 V=800.0 PL=0
MOVL C00545 V=800.0 PL=0
MOVL C00546 V=800.0 PL=0
MOVL C00547 V=800.0 PL=0
MOVL C00548 V=800.0 PL=0
MOVL C00549 V=800.0 PL=0
MOVL C00550 V=800.0 PL=0
MOVL C00551 V=800.0 PL=0
MOVL C00552 V=800.0 PL=0
MOVL C00553 V=800.0 PL=0
MOVL C00554 V=800.0 PL=0
MOVL C00555 V=800.0 PL=0
MOVL C00556 V=800.0 PL=0
MOVL C00557 V=800.0 PL=0
MOVL C00558 V=800.0 PL=0
MOVL C00559 V=800.0 PL=0
MOVL C00560 V=800.0 PL=0
MOVL C00561 V=800.0 PL=0
MOVL C00562 V=800.0 PL=0
MOVL C00563 V=800.0 PL=0
MOVL C00564 V=800.0 PL=0
MOVL C00565 V=800.0 PL=0
MOVL C00566 V=800.0 PL=0
MOVL C00567 V=800.0 PL=0
MOVL C00568 V=800.0 PL=0
MOVL C00569 V=800.0 PL=0
MOVL C00570 V=800.0 PL=0
MOVL C00571 V=800.0 PL=0
MOVL C00572 V=800.0 PL=0
MOVL C00573 V=800.0 PL=0
MOVL C00574 V=800.0 PL=0
MOVL C00575 V=800.0 PL=0
MOVL C00576 V=800.0 PL=0
MOVL C00577 V=800.0 PL=0
MOVL C00578 V=800.0 PL=0
MOVL C00579 V=800.0 PL=0
MOVL C00580 V=800.0 PL=0
MOVL C00581 V=800.0 PL=0
MOVL C00582 V=800.0 PL=0
MOVL C00583 V=800.0 PL=0
MOVL C00584 V=800.0 PL=0
MOVL C00585 V=800.0 PL=0
MOVL C00586 V=800.0 PL=0
MOVL C00587 V=800.0 PL=0
MOVL C00588 V=800.0 PL=0
MOVL C00589 V=800.0 PL=0
MOVL C00590 V=800.0 PL=0
MOVL C00591 V=800.0 PL=0
MOVL C00592 V=800.0 PL=0
MOVL C00593 V=800.0 PL=0
MOVL C00594 V=800.0 PL=0
MOVL C00595 V=800.0 PL=0
MOVL C00596 V=800.0 PL=0
MOVL C00597 V=800.0 PL=0
MOVL C00598 V=800.0 PL=0
MOVL C00599 V=800.0 PL=0
MOVL C00600 V=800.0 PL=0
MOVL C00601 V=800.0 PL=0
MOVL C00602 V=800.0 PL=0
MOVL C00603 V=800.0 PL=0
MOVL C00604 V=800.0 PL=0
MOVL C00605 V=800.0 PL=0
MOVL C00606 V=800.0 PL=0
MOVL C00607 V=800.0 PL=0
MOVL C00608 V=800.0 PL=0
MOVL C00609 V=800.0 PL=0
MOVL C00610 V=800.0 PL=0
MOVL C00611 V=800.0 PL=0
MOVL C00612 V=800.0 PL=0
MOVL C00613 V=800.0 PL=0
MOVL C00614 V=800.0 PL=0
MOVL C00615 V=800.0 PL=0
MOVL C00616 V=800.0 PL=0
MOVL C00617 V=800.0 PL=0
MOVL C00618 V=800.0 PL=0
MOVL C00619 V=800.0 PL=0
MOVL C00620 V=800.0 PL=0
MOVL C00621 V=800.0 PL=0
MOVL C00622 V=800.0 PL=0
MOVL C00623 V=800.0 PL=0
MOVL C00624 V=800.0 PL=0
MOVL C00625 V=800.0 PL=0
MOVL C00626 V=800.0 PL=0
MOVL C00627 V=800.0 PL=0
MOVL C00628 V=800.0 PL=0
MOVL C00629 V=800.0 PL=0
MOVL C00630 V=800.0 PL=0
MOVL C00631 V=800.0 PL=0
MOVL C00632 V=800.0 PL=0
MOVL C00633 V=800.0 PL=0
MOVL C00634 V=800.0 PL=0
MOVL C00635 V=800.0 PL=0
MOVL C00636 V=800.0 PL=0
MOVL C00637 V=800.0 PL=0
MOVL C00638 V=800.0 PL=0
MOVL C00639 V=800.0 PL=0
MOVL C00640 V=800.0 PL=0
MOVL C00641 V=800.0 PL=0
MOVL C00642 V=800.0 PL=0
MOVL C00643 V=800.0 PL=0
MOVL C00644 V=800.0 PL=0
MOVL C00645 V=800.0 PL=0
MOVL C00646 V=800.0 PL=0
MOVL C00647 V=800.0 PL=0
MOVL C00648 V=800.0 PL=0
MOVL C00649 V=800.0 PL=0
MOVL C00650 V=800.0 PL=0
MOVL C00651 V=800.0 PL=0
MOVL C00652 V=800.0 PL=0
MOVL C00653 V=800.0 PL=0
MOVL C00654 V=800.0 PL=0
MOVL C00655 V=800.0 PL=0
MOVL C00656 V=800.0 PL=0
MOVL C00657 V=800.0 PL=0
MOVL C00658 V=800.0 PL=0
MOVL C00659 V=800.0 PL=0
MOVL C00660 V=800.0 PL=0
MOVL C00661 V=800.0 PL=0
MOVL C00662 V=800.0 PL=0
MOVL C00663 V=800.0 PL=0
MOVL C00664 V=800.0 PL=0
MOVL C00665 V=800.0 PL=0
MOVL C00666 V=800.0 PL=0
MOVL C00667 V=800.0 PL=0
MOVL C00668 V=800.0 PL=0
MOVL C00669 V=800.0 PL=0
MOVL C00670 V=800.0 PL=0
MOVL C00671 V=800.0 PL=0
MOVL C00672 V=800.0 PL=0
MOVL C00673 V=800.0 PL=0
MOVL C00674 V=800.0 PL=0
MOVL C00675 V=800.0 PL=0
MOVL C00676 V=800.0 PL=0
MOVL C00677 V=800.0 PL=0
MOVL C00678 V=800.0 PL=0
MOVL C00679 V=800.0 PL=0
MOVL C00680 V=800.0 PL=0
MOVL C00681 V=800.0 PL=0
MOVL C00682 V=800.0 PL=0
MOVL C00683 V=800.0 PL=0
MOVL C00684 V=800.0 PL=0
MOVL C00685 V=800.0 PL=0
MOVL C00686 V=800.0 PL=0
MOVL C00687 V=800.0 PL=0
MOVL C00688 V=800.0 PL=0
MOVL C00689 V=800.0 PL=0
MOVL C00690 V=800.0 PL=0
MOVL C00691 V=800.0 PL=0
MOVL C00692 V=800.0 PL=0
MOVL C00693 V=800.0 PL=0
MOVL C00694 V=800.0 PL=0
MOVL C00695 V=800.0 PL=0
MOVL C00696 V=800.0 PL=0
MOVL C00697 V=800.0 PL=0
MOVL C00698 V=800.0 PL=0
MOVL C00699 V=800.0 PL=0
MOVL C00700 V=800.0 PL=0
MOVL C00701 V=800.0 PL=0
MOVL C00702 V=800.0 PL=0
MOVL C00703 V=800.0 PL=0
MOVL C00704 V=800.0 PL=0
MOVL C00705 V=800.0 PL=0
MOVL C00706 V=800.0 PL=0
MOVL C00707 V=800.0 PL=0
MOVL C00708 V=800.0 PL=0
MOVL C00709 V=800.0 PL=0
MOVL C00710 V=800.0 PL=0
MOVL C00711 V=800.0 PL=0
MOVL C00712 V=800.0 PL=0
MOVL C00713 V=800.0 PL=0
MOVL C00714 V=800.0 PL=0
MOVL C00715 V=800.0 PL=0
MOVL C00716 V=800.0 PL=0
MOVL C00717 V=800.0 PL=0
MOVL C00718 V=800.0 PL=0
MOVL C00719 V=800.0 PL=0
MOVL C00720 V=800.0 PL=0
MOVL C00721 V=800.0 PL=0
MOVL C00722 V=800.0 PL=0
MOVL C00723 V=800.0 PL=0
MOVL C00724 V=800.0 PL=0
MOVL C00725 V=800.0 PL=0
MOVL C00726 V=800.0 PL=0
MOVL C00727 V=800.0 PL=0
MOVL C00728 V=800.0 PL=0
MOVL C00729 V=800.0 PL=0
MOVL C00730 V=800.0 PL=0
MOVL C00731 V=800.0 PL=0
MOVL C00732 V=800.0 PL=0
MOVL C00733 V=800.0 PL=0
MOVL C00734 V=800.0 PL=0
MOVL C00735 V=800.0 PL=0
MOVL C00736 V=800.0 PL=0
MOVL C00737 V=800.0 PL=0
MOVL C00738 V=800.0 PL=0
MOVL C00739 V=800.0 PL=0
MOVL C00740 V=800.0 PL=0
MOVL C00741 V=800.0 PL=0
MOVL C00742 V=800.0 PL=0
MOVL C00743 V=800.0 PL=0
MOVL C00744 V=800.0 PL=0
MOVL C00745 V=800.0 PL=0
MOVL C00746 V=800.0 PL=0
MOVL C00747 V=800.0 PL=0
MOVL C00748 V=800.0 PL=0
MOVL C00749 V=800.0 PL=0
MOVL C00750 V=800.0 PL=0
MOVL C00751 V=800.0 PL=0
MOVL C00752 V=800.0 PL=0
MOVL C00753 V=800.0 PL=0
MOVL C00754 V=800.0 PL=0
MOVL C00755 V=800.0 PL=0
MOVL C00756 V=800.0 PL=0
MOVL C00757 V=800.0 PL=0
MOVL C00758 V=800.0 PL=0
MOVL C00759 V=800.0 PL=0
MOVL C00760 V=800.0 PL=0
MOVL C00761 V=800.0 PL=0
MOVL C00762 V=800.0 PL=0
MOVL C00763 V=800.0 PL=0
MOVL C00764 V=800.0 PL=0
MOVL C00765 V=800.0 PL=0
MOVL C00766 V=800.0 PL=0
MOVL C00767 V=800.0 PL=0
MOVL C00768 V=800.0 PL=0
MOVL C00769 V=800.0 PL=0
MOVL C00770 V=800.0 PL=0
MOVL C00771 V=800.0 PL=0
MOVL C00772 V=800.0 PL=0
MOVL C00773 V=800.0 PL=0
MOVL C00774 V=800.0 PL=0
MOVL C00775 V=800.0 PL=0
MOVL C00776 V=800.0 PL=0
MOVL C00777 V=800.0 PL=0
MOVL C00778 V=800.0 PL=0
MOVL C00779 V=800.0 PL=0
MOVL C00780 V=800.0 PL=0
MOVL C00781 V=800.0 PL=0
MOVL C00782 V=800.0 PL=0
MOVL C00783 V=800.0 PL=0
MOVL C00784 V=800.0 PL=0
MOVL C00785 V=800.0 PL=0
MOVL C00786 V=800.0 PL=0
MOVL C00787 V=800.0 PL=0
MOVL C00788 V=800.0 PL=0
MOVL C00789 V=800.0 PL=0
MOVL C00790 V=800.0 PL=0
MOVL C00791 V=800.0 PL=0
MOVL C00792 V=800.0 PL=0
MOVL C00793 V=800.0 PL=0
MOVL C00794 V=800.0 PL=0
MOVL C00795 V=800.0 PL=0
MOVL C00796 V=800.0 PL=0
MOVL C00797 V=800.0 PL=0
MOVL C00798 V=800.0 PL=0
MOVL C00799 V=800.0 PL=0
MOVL C00800 V=800.0 PL=0
MOVL C00801 V=800.0 PL=0
MOVL C00802 V=800.0 PL=0
MOVL C00803 V=800.0 PL=0
MOVL C00804 V=800.0 PL=0
MOVL C00805 V=800.0 PL=0
MOVL C00806 V=800.0 PL=0
MOVL C00807 V=800.0 PL=0
MOVL C00808 V=800.0 PL=0
MOVL C00809 V=800.0 PL=0
MOVL C00810 V=800.0 PL=0
MOVL C00811 V=800.0 PL=0
MOVL C00812 V=800.0 PL=0
MOVL C00813 V=800.0 PL=0
MOVL C00814 V=800.0 PL=0
MOVL C00815 V=800.0 PL=0
MOVL C00816 V=800.0 PL=0
MOVL C00817 V=800.0 PL=0
MOVL C00818 V=800.0 PL=0
MOVL C00819 V=800.0 PL=0
MOVL C00820 V=800.0 PL=0
MOVL C00821 V=800.0 PL=0
MOVL C00822 V=800.0 PL=0
MOVL C00823 V=800.0 PL=0
MOVL C00824 V=800.0 PL=0
MOVL C00825 V=800.0 PL=0
MOVL C00826 V=800.0 PL=0
MOVL C00827 V=800.0 PL=0
MOVL C00828 V=800.0 PL=0
MOVL C00829 V=800.0 PL=0
MOVL C00830 V=800.0 PL=0
MOVL C00831 V=800.0 PL=0
MOVL C00832 V=800.0 PL=0
MOVL C00833 V=800.0 PL=0
MOVL C00834 V=800.0 PL=0
MOVL C00835 V=800.0 PL=0
MOVL C00836 V=800.0 PL=0
MOVL C00837 V=800.0 PL=0
MOVL C00838 V=800.0 PL=0
MOVL C00839 V=800.0 PL=0
MOVL C00840 V=800.0 PL=0
MOVL C00841 V=800.0 PL=0
MOVL C00842 V=800.0 PL=0
MOVL C00843 V=800.0 PL=0
MOVL C00844 V=800.0 PL=0
MOVL C00845 V=800.0 PL=0
MOVL C00846 V=800.0 PL=0
MOVL C00847 V=800.0 PL=0
MOVL C00848 V=800.0 PL=0
MOVL C00849 V=800.0 PL=0
MOVL C00850 V=800.0 PL=0
MOVL C00851 V=800.0 PL=0
MOVL C00852 V=800.0 PL=0
MOVL C00853 V=800.0 PL=0
MOVL C00854 V=800.0 PL=0
MOVL C00855 V=800.0 PL=0
MOVL C00856 V=800.0 PL=0
MOVL C00857 V=800.0 PL=0
MOVL C00858 V=800.0 PL=0
MOVL C00859 V=800.0 PL=0
MOVL C00860 V=800.0 PL=0
MOVL C00861 V=800.0 PL=0
MOVL C00862 V=800.0 PL=0
MOVL C00863 V=800.0 PL=0
MOVL C00864 V=800.0 PL=0
MOVL C00865 V=800.0 PL=0
MOVL C00866 V=800.0 PL=0
MOVL C00867 V=800.0 PL=0
MOVL C00868 V=800.0 PL=0
MOVL C00869 V=800.0 PL=0
MOVL C00870 V=800.0 PL=0
MOVL C00871 V=800.0 PL=0
MOVL C00872 V=800.0 PL=0
MOVL C00873 V=800.0 PL=0
MOVL C00874 V=800.0 PL=0
MOVL C00875 V=800.0 PL=0
MOVL C00876 V=800.0 PL=0
MOVL C00877 V=800.0 PL=0
MOVL C00878 V=800.0 PL=0
MOVL C00879 V=800.0 PL=0
MOVL C00880 V=800.0 PL=0
MOVL C00881 V=800.0 PL=0
MOVL C00882 V=800.0 PL=0
MOVL C00883 V=800.0 PL=0
MOVL C00884 V=800.0 PL=0
MOVL C00885 V=800.0 PL=0
MOVL C00886 V=800.0 PL=0
MOVL C00887 V=800.0 PL=0
MOVL C00888 V=800.0 PL=0
MOVL C00889 V=800.0 PL=0
MOVL C00890 V=800.0 PL=0
MOVL C00891 V=800.0 PL=0
MOVL C00892 V=800.0 PL=0
MOVL C00893 V=800.0 PL=0
MOVL C00894 V=800.0 PL=0
MOVL C00895 V=800.0 PL=0
MOVL C00896 V=800.0 PL=0
MOVL C00897 V=800.0 PL=0
MOVL C00898 V=800.0 PL=0
MOVL C00899 V=800.0 PL=0
MOVL C00900 V=800.0 PL=0
MOVL C00901 V=800.0 PL=0
MOVL C00902 V=800.0 PL=0
MOVL C00903 V=800.0 PL=0
MOVL C00904 V=800.0 PL=0
MOVL C00905 V=800.0 PL=0
MOVL C00906 V=800.0 PL=0
MOVL C00907 V=800.0 PL=0
MOVL C00908 V=800.0 PL=0
MOVL C00909 V=800.0 PL=0
MOVL C00910 V=800.0 PL=0
MOVL C00911 V=800.0 PL=0
MOVL C00912 V=800.0 PL=0
MOVL C00913 V=800.0 PL=0
MOVL C00914 V=800.0 PL=0
MOVL C00915 V=800.0 PL=0
MOVL C00916 V=800.0 PL=0
MOVL C00917 V=800.0 PL=0
MOVL C00918 V=800.0 PL=0
MOVL C00919 V=800.0 PL=0
MOVL C00920 V=800.0 PL=0
MOVL C00921 V=800.0 PL=0
MOVL C00922 V=800.0 PL=0
MOVL C00923 V=800.0 PL=0
MOVL C00924 V=800.0 PL=0
MOVL C00925 V=800.0 PL=0
MOVL C00926 V=800.0 PL=0
MOVL C00927 V=800.0 PL=0
MOVL C00928 V=800.0 PL=0
MOVL C00929 V=800.0 PL=0
MOVL C00930 V=800.0 PL=0
MOVL C00931 V=800.0 PL=0
MOVL C00932 V=800.0 PL=0
MOVL C00933 V=800.0 PL=0
MOVL C00934 V=800.0 PL=0
MOVL C00935 V=800.0 PL=0
MOVL C00936 V=800.0 PL=0
MOVL C00937 V=800.0 PL=0
MOVL C00938 V=800.0 PL=0
MOVL C00939 V=800.0 PL=0
MOVL C00940 V=800.0 PL=0
MOVL C00941 V=800.0 PL=0
MOVL C00942 V=800.0 PL=0
MOVL C00943 V=800.0 PL=0
MOVL C00944 V=800.0 PL=0
MOVL C00945 V=800.0 PL=0
MOVL C00946 V=800.0 PL=0
MOVL C00947 V=800.0 PL=0
MOVL C00948 V=800.0 PL=0
MOVL C00949 V=800.0 PL=0
MOVL C00950 V=800.0 PL=0
MOVL C00951 V=800.0 PL=0
MOVL C00952 V=800.0 PL=0
MOVL C00953 V=800.0 PL=0
MOVL C00954 V=800.0 PL=0
MOVL C00955 V=800.0 PL=0
MOVL C00956 V=800.0 PL=0
MOVL C00957 V=800.0 PL=0
MOVL C00958 V=800.0 PL=0
MOVL C00959 V=800.0 PL=0
MOVL C00960 V=800.0 PL=0
MOVL C00961 V=800.0 PL=0
MOVL C00962 V=800.0 PL=0
MOVL C00963 V=800.0 PL=0
MOVL C00964 V=800.0 PL=0
MOVL C00965 V=800.0 PL=0
MOVL C00966 V=800.0 PL=0
MOVL C00967 V=800.0 PL=0
MOVL C00968 V=800.0 PL=0
MOVL C00969 V=800.0 PL=0
MOVL C00970 V=800.0 PL=0
MOVL C00971 V=800.0 PL=0
MOVL C00972 V=800.0 PL=0
MOVL C00973 V=800.0 PL=0
MOVL C00974 V=800.0 PL=0
MOVL C00975 V=800.0 PL=0
MOVL C00976 V=800.0 PL=0
MOVL C00977 V=800.0 PL=0
MOVL C00978 V=800.0 PL=0
MOVL C00979 V=800.0 PL=0
MOVL C00980 V=800.0 PL=0
MOVL C00981 V=800.0 PL=0
MOVL C00982 V=800.0 PL=0
MOVL C00983 V=800.0 PL=0
MOVL C00984 V=800.0 PL=0
MOVL C00985 V=800.0 PL=0
MOVL C00986 V=800.0 PL=0
MOVL C00987 V=800.0 PL=0
MOVL C00988 V=800.0 PL=0
MOVL C00989 V=800.0 PL=0
MOVL C00990 V=800.0 PL=0
MOVL C00991 V=800.0 PL=0
MOVL C00992 V=800.0 PL=0
MOVL C00993 V=800.0 PL=0
MOVL C00994 V=800.0 PL=0
MOVL C00995 V=800.0 PL=0
MOVL C00996 V=800.0 PL=0
MOVL C00997 V=800.0 PL=0
MOVL C00998 V=800.0 PL=0
MOVL C00999 V=800.0 PL=0
MOVL C01000 V=800.0 PL=0
MOVL C01001 V=800.0 PL=0
MOVL C01002 V=800.0 PL=0
MOVL C01003 V=800.0 PL=0
MOVL C01004 V=800.0 PL=0
MOVL C01005 V=800.0 PL=0
MOVL C01006 V=800.0 PL=0
MOVL C01007 V=800.0 PL=0
MOVL C01008 V=800.0 PL=0
MOVL C01009 V=800.0 PL=0
MOVL C01010 V=800.0 PL=0
MOVL C01011 V=800.0 PL=0
MOVL C01012 V=800.0 PL=0
MOVL C01013 V=800.0 PL=0
MOVL C01014 V=800.0 PL=0
MOVL C01015 V=800.0 PL=0
MOVL C01016 V=800.0 PL=0
MOVL C01017 V=800.0 PL=0
MOVL C01018 V=800.0 PL=0
MOVL C01019 V=800.0 PL=0
MOVL C01020 V=800.0 PL=0
MOVL C01021 V=800.0 PL=0
MOVL C01022 V=800.0 PL=0
MOVL C01023 V=800.0 PL=0
MOVL C01024 V=800.0 PL=0
MOVL C01025 V=800.0 PL=0
MOVL C01026 V=800.0 PL=0
MOVL C01027 V=800.0 PL=0
MOVL C01028 V=800.0 PL=0
MOVL C01029 V=800.0 PL=0
MOVL C01030 V=800.0 PL=0
MOVL C01031 V=800.0 PL=0
MOVL C01032 V=800.0 PL=0
MOVL C01033 V=800.0 PL=0
MOVL C01034 V=800.0 PL=0
MOVL C01035 V=800.0 PL=0
MOVL C01036 V=800.0 PL=0
MOVL C01037 V=800.0 PL=0
MOVL C01038 V=800.0 PL=0
MOVL C01039 V=800.0 PL=0
MOVL C01040 V=800.0 PL=0
MOVL C01041 V=800.0 PL=0
MOVL C01042 V=800.0 PL=0
MOVL C01043 V=800.0 PL=0
MOVL C01044 V=800.0 PL=0
MOVL C01045 V=800.0 PL=0
MOVL C01046 V=800.0 PL=0
MOVL C01047 V=800.0 PL=0
MOVL C01048 V=800.0 PL=0
MOVL C01049 V=800.0 PL=0
MOVL C01050 V=800.0 PL=0
MOVL C01051 V=800.0 PL=0
MOVL C01052 V=800.0 PL=0
MOVL C01053 V=800.0 PL=0
MOVL C01054 V=800.0 PL=0
MOVL C01055 V=800.0 PL=0
MOVL C01056 V=800.0 PL=0
MOVL C01057 V=800.0 PL=0
MOVL C01058 V=800.0 PL=0
MOVL C01059 V=800.0 PL=0
MOVL C01060 V=800.0 PL=0
MOVL C01061 V=800.0 PL=0
MOVL C01062 V=800.0 PL=0
MOVL C01063 V=800.0 PL=0
MOVL C01064 V=800.0 PL=0
MOVL C01065 V=800.0 PL=0
MOVL C01066 V=800.0 PL=0
MOVL C01067 V=800.0 PL=0
MOVL C01068 V=800.0 PL=0
MOVL C01069 V=800.0 PL=0
MOVL C01070 V=800.0 PL=0
MOVL C01071 V=800.0 PL=0
MOVL C01072 V=800.0 PL=0
MOVL C01073 V=800.0 PL=0
MOVL C01074 V=800.0 PL=0
MOVL C01075 V=800.0 PL=0
MOVL C01076 V=800.0 PL=0
MOVL C01077 V=800.0 PL=0
MOVL C01078 V=800.0 PL=0
MOVL C01079 V=800.0 PL=0
MOVL C01080 V=800.0 PL=0
MOVL C01081 V=800.0 PL=0
MOVL C01082 V=800.0 PL=0
MOVL C01083 V=800.0 PL=0
MOVL C01084 V=800.0 PL=0
MOVL C01085 V=800.0 PL=0
MOVL C01086 V=800.0 PL=0
MOVL C01087 V=800.0 PL=0
MOVL C01088 V=800.0 PL=0
MOVL C01089 V=800.0 PL=0
MOVL C01090 V=800.0 PL=0
MOVL C01091 V=800.0 PL=0
MOVL C01092 V=800.0 PL=0
MOVL C01093 V=800.0 PL=0
MOVL C01094 V=800.0 PL=0
MOVL C01095 V=800.0 PL=0
MOVL C01096 V=800.0 PL=0
MOVL C01097 V=800.0 PL=0
MOVL C01098 V=800.0 PL=0
MOVL C01099 V=800.0 PL=0
MOVL C01100 V=800.0 PL=0
MOVL C01101 V=800.0 PL=0
MOVL C01102 V=800.0 PL=0
MOVL C01103 V=800.0 PL=0
MOVL C01104 V=800.0 PL=0
MOVL C01105 V=800.0 PL=0
MOVL C01106 V=800.0 PL=0
MOVL C01107 V=800.0 PL=0
MOVL C01108 V=800.0 PL=0
MOVL C01109 V=800.0 PL=0
MOVL C01110 V=800.0 PL=0
MOVL C01111 V=800.0 PL=0
MOVL C01112 V=800.0 PL=0
MOVL C01113 V=800.0 PL=0
MOVL C01114 V=800.0 PL=0
MOVL C01115 V=800.0 PL=0
MOVL C01116 V=800.0 PL=0
MOVL C01117 V=800.0 PL=0
MOVL C01118 V=800.0 PL=0
MOVL C01119 V=800.0 PL=0
MOVL C01120 V=800.0 PL=0
MOVL C01121 V=800.0 PL=0
MOVL C01122 V=800.0 PL=0
MOVL C01123 V=800.0 PL=0
MOVL C01124 V=800.0 PL=0
MOVL C01125 V=800.0 PL=0
MOVL C01126 V=800.0 PL=0
MOVL C01127 V=800.0 PL=0
MOVL C01128 V=800.0 PL=0
MOVL C01129 V=800.0 PL=0
MOVL C01130 V=800.0 PL=0
MOVL C01131 V=800.0 PL=0
MOVL C01132 V=800.0 PL=0
MOVL C01133 V=800.0 PL=0
MOVL C01134 V=800.0 PL=0
MOVL C01135 V=800.0 PL=0
MOVL C01136 V=800.0 PL=0
MOVL C01137 V=800.0 PL=0
MOVL C01138 V=800.0 PL=0
MOVL C01139 V=800.0 PL=0
MOVL C01140 V=800.0 PL=0
MOVL C01141 V=800.0 PL=0
MOVL C01142 V=800.0 PL=0
MOVL C01143 V=800.0 PL=0
MOVL C01144 V=800.0 PL=0
MOVL C01145 V=800.0 PL=0
MOVL C01146 V=800.0 PL=0
MOVL C01147 V=800.0 PL=0
MOVL C01148 V=800.0 PL=0
MOVL C01149 V=800.0 PL=0
MOVL C01150 V=800.0 PL=0
MOVL C01151 V=800.0 PL=0
MOVL C01152 V=800.0 PL=0
MOVL C01153 V=800.0 PL=0
MOVL C01154 V=800.0 PL=0
MOVL C01155 V=800.0 PL=0
MOVL C01156 V=800.0 PL=0
MOVL C01157 V=800.0 PL=0
MOVL C01158 V=800.0 PL=0
MOVL C01159 V=800.0 PL=0
MOVL C01160 V=800.0 PL=0
MOVL C01161 V=800.0 PL=0
MOVL C01162 V=800.0 PL=0
MOVL C01163 V=800.0 PL=0
MOVL C01164 V=800.0 PL=0
MOVL C01165 V=800.0 PL=0
MOVL C01166 V=800.0 PL=0
MOVL C01167 V=800.0 PL=0
MOVL C01168 V=800.0 PL=0
MOVL C01169 V=800.0 PL=0
MOVL C01170 V=800.0 PL=0
MOVL C01171 V=800.0 PL=0
MOVL C01172 V=800.0 PL=0
MOVL C01173 V=800.0 PL=0
MOVL C01174 V=800.0 PL=0
MOVL C01175 V=800.0 PL=0
MOVL C01176 V=800.0 PL=0
MOVL C01177 V=800.0 PL=0
MOVL C01178 V=800.0 PL=0
MOVL C01179 V=800.0 PL=0
MOVL C01180 V=800.0 PL=0
MOVL C01181 V=800.0 PL=0
MOVL C01182 V=800.0 PL=0
MOVL C01183 V=800.0 PL=0
MOVL C01184 V=800.0 PL=0
MOVL C01185 V=800.0 PL=0
MOVL C01186 V=800.0 PL=0
MOVL C01187 V=800.0 PL=0
MOVL C01188 V=800.0 PL=0
MOVL C01189 V=800.0 PL=0
MOVL C01190 V=800.0 PL=0
MOVL C01191 V=800.0 PL=0
MOVL C01192 V=800.0 PL=0
MOVL C01193 V=800.0 PL=0
MOVL C01194 V=800.0 PL=0
MOVL C01195 V=800.0 PL=0
MOVL C01196 V=800.0 PL=0
MOVL C01197 V=800.0 PL=0
MOVL C01198 V=800.0 PL=0
MOVL C01199 V=800.0 PL=0
MOVL C01200 V=800.0 PL=0
MOVL C01201 V=800.0 PL=0
MOVL C01202 V=800.0 PL=0
MOVL C01203 V=800.0 PL=0
MOVL C01204 V=800.0 PL=0
MOVL C01205 V=800.0 PL=0
MOVL C01206 V=800.0 PL=0
MOVL C01207 V=800.0 PL=0
MOVL C01208 V=800.0 PL=0
MOVL C01209 V=800.0 PL=0
MOVL C01210 V=800.0 PL=0
MOVL C01211 V=800.0 PL=0
MOVL C01212 V=800.0 PL=0
MOVL C01213 V=800.0 PL=0
MOVL C01214 V=800.0 PL=0
MOVL C01215 V=800.0 PL=0
MOVL C01216 V=800.0 PL=0
MOVL C01217 V=800.0 PL=0
MOVL C01218 V=800.0 PL=0
MOVL C01219 V=800.0 PL=0
MOVL C01220 V=800.0 PL=0
MOVL C01221 V=800.0 PL=0
MOVL C01222 V=800.0 PL=0
MOVL C01223 V=800.0 PL=0
MOVL C01224 V=800.0 PL=0
MOVL C01225 V=800.0 PL=0
MOVL C01226 V=800.0 PL=0
MOVL C01227 V=800.0 PL=0
MOVL C01228 V=800.0 PL=0
MOVL C01229 V=800.0 PL=0
MOVL C01230 V=800.0 PL=0
MOVL C01231 V=800.0 PL=0
MOVL C01232 V=800.0 PL=0
MOVL C01233 V=800.0 PL=0
MOVL C01234 V=800.0 PL=0
MOVL C01235 V=800.0 PL=0
MOVL C01236 V=800.0 PL=0
MOVL C01237 V=800.0 PL=0
MOVL C01238 V=800.0 PL=0
MOVL C01239 V=800.0 PL=0
MOVL C01240 V=800.0 PL=0
MOVL C01241 V=800.0 PL=0
MOVL C01242 V=800.0 PL=0
MOVL C01243 V=800.0 PL=0
MOVL C01244 V=800.0 PL=0
MOVL C01245 V=800.0 PL=0
MOVL C01246 V=800.0 PL=0
MOVL C01247 V=800.0 PL=0
MOVL C01248 V=800.0 PL=0
MOVL C01249 V=800.0 PL=0
MOVL C01250 V=800.0 PL=0
MOVL C01251 V=800.0 PL=0
MOVL C01252 V=800.0 PL=0
MOVL C01253 V=800.0 PL=0
MOVL C01254 V=800.0 PL=0
MOVL C01255 V=800.0 PL=0
MOVL C01256 V=800.0 PL=0
MOVL C01257 V=800.0 PL=0
MOVL C01258 V=800.0 PL=0
MOVL C01259 V=800.0 PL=0
MOVL C01260 V=800.0 PL=0
MOVL C01261 V=800.0 PL=0
MOVL C01262 V=800.0 PL=0
MOVL C01263 V=800.0 PL=0
MOVL C01264 V=800.0 PL=0
MOVL C01265 V=800.0 PL=0
MOVL C01266 V=800.0 PL=0
MOVL C01267 V=800.0 PL=0
MOVL C01268 V=800.0 PL=0
MOVL C01269 V=800.0 PL=0
MOVL C01270 V=800.0 PL=0
MOVL C01271 V=800.0 PL=0
MOVL C01272 V=800.0 PL=0
MOVL C01273 V=800.0 PL=0
MOVL C01274 V=800.0 PL=0
MOVL C01275 V=800.0 PL=0
MOVL C01276 V=800.0 PL=0
MOVL C01277 V=800.0 PL=0
MOVL C01278 V=800.0 PL=0
MOVL C01279 V=800.0 PL=0
MOVL C01280 V=800.0 PL=0
MOVL C01281 V=800.0 PL=0
MOVL C01282 V=800.0 PL=0
MOVL C01283 V=800.0 PL=0
MOVL C01284 V=800.0 PL=0
MOVL C01285 V=800.0 PL=0
MOVL C01286 V=800.0 PL=0
MOVL C01287 V=800.0 PL=0
MOVL C01288 V=800.0 PL=0
MOVL C01289 V=800.0 PL=0
MOVL C01290 V=800.0 PL=0
MOVL C01291 V=800.0 PL=0
MOVL C01292 V=800.0 PL=0
MOVL C01293 V=800.0 PL=0
MOVL C01294 V=800.0 PL=0
MOVL C01295 V=800.0 PL=0
MOVL C01296 V=800.0 PL=0
MOVL C01297 V=800.0 PL=0
MOVL C01298 V=800.0 PL=0
MOVL C01299 V=800.0 PL=0
MOVL C01300 V=800.0 PL=0
MOVL C01301 V=800.0 PL=0
MOVL C01302 V=800.0 PL=0
MOVL C01303 V=800.0 PL=0
MOVL C01304 V=800.0 PL=0
MOVL C01305 V=800.0 PL=0
MOVL C01306 V=800.0 PL=0
MOVL C01307 V=800.0 PL=0
MOVL C01308 V=800.0 PL=0
MOVL C01309 V=800.0 PL=0
MOVL C01310 V=800.0 PL=0
MOVL C01311 V=800.0 PL=0
MOVL C01312 V=800.0 PL=0
MOVL C01313 V=800.0 PL=0
MOVL C01314 V=800.0 PL=0
MOVL C01315 V=800.0 PL=0
MOVL C01316 V=800.0 PL=0
MOVL C01317 V=800.0 PL=0
MOVL C01318 V=800.0 PL=0
MOVL C01319 V=800.0 PL=0
MOVL C01320 V=800.0 PL=0
MOVL C01321 V=800.0 PL=0
MOVL C01322 V=800.0 PL=0
MOVL C01323 V=800.0 PL=0
MOVL C01324 V=800.0 PL=0
MOVL C01325 V=800.0 PL=0
MOVL C01326 V=800.0 PL=0
MOVL C01327 V=800.0 PL=0
MOVL C01328 V=800.0 PL=0
MOVL C01329 V=800.0 PL=0
MOVL C01330 V=800.0 PL=0
MOVL C01331 V=800.0 PL=0
MOVL C01332 V=800.0 PL=0
MOVL C01333 V=800.0 PL=0
MOVL C01334 V=800.0 PL=0
MOVL C01335 V=800.0 PL=0
MOVL C01336 V=800.0 PL=0
MOVL C01337 V=800.0 PL=0
MOVL C01338 V=800.0 PL=0
MOVL C01339 V=800.0 PL=0
MOVL C01340 V=800.0 PL=0
MOVL C01341 V=800.0 PL=0
MOVL C01342 V=800.0 PL=0
MOVL C01343 V=800.0 PL=0
MOVL C01344 V=800.0 PL=0
MOVL C01345 V=800.0 PL=0
MOVL C01346 V=800.0 PL=0
MOVL C01347 V=800.0 PL=0
MOVL C01348 V=800.0 PL=0
MOVL C01349 V=800.0 PL=0
MOVL C01350 V=800.0 PL=0
MOVL C01351 V=800.0 PL=0
MOVL C01352 V=800.0 PL=0
MOVL C01353 V=800.0 PL=0
MOVL C01354 V=800.0 PL=0
MOVL C01355 V=800.0 PL=0
MOVL C01356 V=800.0 PL=0
MOVL C01357 V=800.0 PL=0
MOVL C01358 V=800.0 PL=0
MOVL C01359 V=800.0 PL=0
MOVL C01360 V=800.0 PL=0
MOVL C01361 V=800.0 PL=0
MOVL C01362 V=800.0 PL=0
MOVL C01363 V=800.0 PL=0
MOVL C01364 V=800.0 PL=0
MOVL C01365 V=800.0 PL=0
MOVL C01366 V=800.0 PL=0
MOVL C01367 V=800.0 PL=0
MOVL C01368 V=800.0 PL=0
MOVL C01369 V=800.0 PL=0
MOVL C01370 V=800.0 PL=0
MOVL C01371 V=800.0 PL=0
MOVL C01372 V=800.0 PL=0
MOVL C01373 V=800.0 PL=0
MOVL C01374 V=800.0 PL=0
MOVL C01375 V=800.0 PL=0
MOVL C01376 V=800.0 PL=0
MOVL C01377 V=800.0 PL=0
MOVL C01378 V=800.0 PL=0
MOVL C01379 V=800.0 PL=0
MOVL C01380 V=800.0 PL=0
MOVL C01381 V=800.0 PL=0
MOVL C01382 V=800.0 PL=0
MOVL C01383 V=800.0 PL=0
MOVL C01384 V=800.0 PL=0
MOVL C01385 V=800.0 PL=0
MOVL C01386 V=800.0 PL=0
MOVL C01387 V=800.0 PL=0
MOVL C01388 V=800.0 PL=0
MOVL C01389 V=800.0 PL=0
MOVL C01390 V=800.0 PL=0
MOVL C01391 V=800.0 PL=0
MOVL C01392 V=800.0 PL=0
MOVL C01393 V=800.0 PL=0
MOVL C01394 V=800.0 PL=0
MOVL C01395 V=800.0 PL=0
MOVL C01396 V=800.0 PL=0
MOVL C01397 V=800.0 PL=0
MOVL C01398 V=800.0 PL=0
MOVL C01399 V=800.0 PL=0
MOVL C01400 V=800.0 PL=0
MOVL C01401 V=800.0 PL=0
MOVL C01402 V=800.0 PL=0
MOVL C01403 V=800.0 PL=0
MOVL C01404 V=800.0 PL=0
MOVL C01405 V=800.0 PL=0
MOVL C01406 V=800.0 PL=0
MOVL C01407 V=800.0 PL=0
MOVL C01408 V=800.0 PL=0
MOVL C01409 V=800.0 PL=0
MOVL C01410 V=800.0 PL=0
MOVL C01411 V=800.0 PL=0
MOVL C01412 V=800.0 PL=0
MOVL C01413 V=800.0 PL=0
MOVL C01414 V=800.0 PL=0
MOVL C01415 V=800.0 PL=0
MOVL C01416 V=800.0 PL=0
MOVL C01417 V=800.0 PL=0
MOVL C01418 V=800.0 PL=0
MOVL C01419 V=800.0 PL=0
MOVL C01420 V=800.0 PL=0
MOVL C01421 V=800.0 PL=0
MOVL C01422 V=800.0 PL=0
MOVL C01423 V=800.0 PL=0
MOVL C01424 V=800.0 PL=0
MOVL C01425 V=800.0 PL=0
MOVL C01426 V=800.0 PL=0
MOVL C01427 V=800.0 PL=0
MOVL C01428 V=800.0 PL=0
MOVL C01429 V=800.0 PL=0
MOVL C01430 V=800.0 PL=0
MOVL C01431 V=800.0 PL=0
MOVL C01432 V=800.0 PL=0
MOVL C01433 V=800.0 PL=0
MOVL C01434 V=800.0 PL=0
MOVL C01435 V=800.0 PL=0
MOVL C01436 V=800.0 PL=0
MOVL C01437 V=800.0 PL=0
MOVL C01438 V=800.0 PL=0
MOVL C01439 V=800.0 PL=0
MOVL C01440 V=800.0 PL=0
MOVL C01441 V=800.0 PL=0
MOVL C01442 V=800.0 PL=0
MOVL C01443 V=800.0 PL=0
MOVL C01444 V=800.0 PL=0
MOVL C01445 V=800.0 PL=0
MOVL C01446 V=800.0 PL=0
MOVL C01447 V=800.0 PL=0
MOVL C01448 V=800.0 PL=0
MOVL C01449 V=800.0 PL=0
MOVL C01450 V=800.0 PL=0
MOVL C01451 V=800.0 PL=0
MOVL C01452 V=800.0 PL=0
MOVL C01453 V=800.0 PL=0
MOVL C01454 V=800.0 PL=0
MOVL C01455 V=800.0 PL=0
MOVL C01456 V=800.0 PL=0
MOVL C01457 V=800.0 PL=0
MOVL C01458 V=800.0 PL=0
MOVL C01459 V=800.0 PL=0
MOVL C01460 V=800.0 PL=0
MOVL C01461 V=800.0 PL=0
MOVL C01462 V=800.0 PL=0
MOVL C01463 V=800.0 PL=0
MOVL C01464 V=800.0 PL=0
MOVL C01465 V=800.0 PL=0
MOVL C01466 V=800.0 PL=0
MOVL C01467 V=800.0 PL=0
MOVL C01468 V=800.0 PL=0
MOVL C01469 V=800.0 PL=0
MOVL C01470 V=800.0 PL=0
MOVL C01471 V=800.0 PL=0
MOVL C01472 V=800.0 PL=0
MOVL C01473 V=800.0 PL=0
MOVL C01474 V=800.0 PL=0
MOVL C01475 V=800.0 PL=0
MOVL C01476 V=800.0 PL=0
MOVL C01477 V=800.0 PL=0
MOVL C01478 V=800.0 PL=0
MOVL C01479 V=800.0 PL=0
MOVL C01480 V=800.0 PL=0
MOVL C01481 V=800.0 PL=0
MOVL C01482 V=800.0 PL=0
MOVL C01483 V=800.0 PL=0
MOVL C01484 V=800.0 PL=0
MOVL C01485 V=800.0 PL=0
MOVL C01486 V=800.0 PL=0
MOVL C01487 V=800.0 PL=0
MOVL C01488 V=800.0 PL=0
MOVL C01489 V=800.0 PL=0
MOVL C01490 V=800.0 PL=0
MOVL C01491 V=800.0 PL=0
MOVL C01492 V=800.0 PL=0
MOVL C01493 V=800.0 PL=0
MOVL C01494 V=800.0 PL=0
MOVL C01495 V=800.0 PL=0
MOVL C01496 V=800.0 PL=0
MOVL C01497 V=800.0 PL=0
MOVL C01498 V=800.0 PL=0
MOVL C01499 V=800.0 PL=0
MOVL C01500 V=800.0 PL=0
MOVL C01501 V=800.0 PL=0
MOVL C01502 V=800.0 PL=0
MOVL C01503 V=800.0 PL=0
MOVL C01504 V=800.0 PL=0
MOVL C01505 V=800.0 PL=0
MOVL C01506 V=800.0 PL=0
MOVL C01507 V=800.0 PL=0
MOVL C01508 V=800.0 PL=0
MOVL C01509 V=800.0 PL=0
MOVL C01510 V=800.0 PL=0
MOVL C01511 V=800.0 PL=0
MOVL C01512 V=800.0 PL=0
MOVL C01513 V=800.0 PL=0
MOVL C01514 V=800.0 PL=0
MOVL C01515 V=800.0 PL=0
MOVL C01516 V=800.0 PL=0
MOVL C01517 V=800.0 PL=0
MOVL C01518 V=800.0 PL=0
MOVL C01519 V=800.0 PL=0
MOVL C01520 V=800.0 PL=0
MOVL C01521 V=800.0 PL=0
MOVL C01522 V=800.0 PL=0
MOVL C01523 V=800.0 PL=0
MOVL C01524 V=800.0 PL=0
MOVL C01525 V=800.0 PL=0
MOVL C01526 V=800.0 PL=0
MOVL C01527 V=800.0 PL=0
MOVL C01528 V=800.0 PL=0
MOVL C01529 V=800.0 PL=0
MOVL C01530 V=800.0 PL=0
MOVL C01531 V=800.0 PL=0
MOVL C01532 V=800.0 PL=0
MOVL C01533 V=800.0 PL=0
MOVL C01534 V=800.0 PL=0
MOVL C01535 V=800.0 PL=0
MOVL C01536 V=800.0 PL=0
MOVL C01537 V=800.0 PL=0
MOVL C01538 V=800.0 PL=0
MOVL C01539 V=800.0 PL=0
MOVL C01540 V=800.0 PL=0
MOVL C01541 V=800.0 PL=0
MOVL C01542 V=800.0 PL=0
MOVL C01543 V=800.0 PL=0
MOVL C01544 V=800.0 PL=0
MOVL C01545 V=800.0 PL=0
MOVL C01546 V=800.0 PL=0
MOVL C01547 V=800.0 PL=0
MOVL C01548 V=800.0 PL=0
MOVL C01549 V=800.0 PL=0
MOVL C01550 V=800.0 PL=0
MOVL C01551 V=800.0 PL=0
MOVL C01552 V=800.0 PL=0
MOVL C01553 V=800.0 PL=0
MOVL C01554 V=800.0 PL=0
MOVL C01555 V=800.0 PL=0
MOVL C01556 V=800.0 PL=0
MOVL C01557 V=800.0 PL=0
MOVL C01558 V=800.0 PL=0
MOVL C01559 V=800.0 PL=0
MOVL C01560 V=800.0 PL=0
MOVL C01561 V=800.0 PL=0
MOVL C01562 V=800.0 PL=0
MOVL C01563 V=800.0 PL=0
MOVL C01564 V=800.0 PL=0
MOVL C01565 V=800.0 PL=0
MOVL C01566 V=800.0 PL=0
MOVL C01567 V=800.0 PL=0
MOVL C01568 V=800.0 PL=0
MOVL C01569 V=800.0 PL=0
MOVL C01570 V=800.0 PL=0
MOVL C01571 V=800.0 PL=0
MOVL C01572 V=800.0 PL=0
MOVL C01573 V=800.0 PL=0
MOVL C01574 V=800.0 PL=0
MOVL C01575 V=800.0 PL=0
MOVL C01576 V=800.0 PL=0
MOVL C01577 V=800.0 PL=0
MOVL C01578 V=800.0 PL=0
MOVL C01579 V=800.0 PL=0
MOVL C01580 V=800.0 PL=0
MOVL C01581 V=800.0 PL=0
MOVL C01582 V=800.0 PL=0
MOVL C01583 V=800.0 PL=0
MOVL C01584 V=800.0 PL=0
MOVL C01585 V=800.0 PL=0
MOVL C01586 V=800.0 PL=0
MOVL C01587 V=800.0 PL=0
MOVL C01588 V=800.0 PL=0
MOVL C01589 V=800.0 PL=0
MOVL C01590 V=800.0 PL=0
MOVL C01591 V=800.0 PL=0
MOVL C01592 V=800.0 PL=0
MOVL C01593 V=800.0 PL=0
MOVL C01594 V=800.0 PL=0
MOVL C01595 V=800.0 PL=0
MOVL C01596 V=800.0 PL=0
MOVL C01597 V=800.0 PL=0
MOVL C01598 V=800.0 PL=0
MOVL C01599 V=800.0 PL=0
MOVL C01600 V=800.0 PL=0
MOVL C01601 V=800.0 PL=0
MOVL C01602 V=800.0 PL=0
MOVL C01603 V=800.0 PL=0
MOVL C01604 V=800.0 PL=0
MOVL C01605 V=800.0 PL=0
MOVL C01606 V=800.0 PL=0
MOVL C01607 V=800.0 PL=0
MOVL C01608 V=800.0 PL=0
MOVL C01609 V=800.0 PL=0
MOVL C01610 V=800.0 PL=0
MOVL C01611 V=800.0 PL=0
MOVL C01612 V=800.0 PL=0
MOVL C01613 V=800.0 PL=0
MOVL C01614 V=800.0 PL=0
MOVL C01615 V=800.0 PL=0
MOVL C01616 V=800.0 PL=0
MOVL C01617 V=800.0 PL=0
MOVL C01618 V=800.0 PL=0
MOVL C01619 V=800.0 PL=0
MOVL C01620 V=800.0 PL=0
MOVL C01621 V=800.0 PL=0
MOVL C01622 V=800.0 PL=0
MOVL C01623 V=800.0 PL=0
MOVL C01624 V=800.0 PL=0
MOVL C01625 V=800.0 PL=0
MOVL C01626 V=800.0 PL=0
MOVL C01627 V=800.0 PL=0
MOVL C01628 V=800.0 PL=0
MOVL C01629 V=800.0 PL=0
MOVL C01630 V=800.0 PL=0
MOVL C01631 V=800.0 PL=0
MOVL C01632 V=800.0 PL=0
MOVL C01633 V=800.0 PL=0
MOVL C01634 V=800.0 PL=0
MOVL C01635 V=800.0 PL=0
MOVL C01636 V=800.0 PL=0
MOVL C01637 V=800.0 PL=0
MOVL C01638 V=800.0 PL=0
MOVL C01639 V=800.0 PL=0
MOVL C01640 V=800.0 PL=0
MOVL C01641 V=800.0 PL=0
MOVL C01642 V=800.0 PL=0
MOVL C01643 V=800.0 PL=0
MOVL C01644 V=800.0 PL=0
MOVL C01645 V=800.0 PL=0
MOVL C01646 V=800.0 PL=0
MOVL C01647 V=800.0 PL=0
MOVL C01648 V=800.0 PL=0
MOVL C01649 V=800.0 PL=0
MOVL C01650 V=800.0 PL=0
MOVL C01651 V=800.0 PL=0
MOVL C01652 V=800.0 PL=0
MOVL C01653 V=800.0 PL=0
MOVL C01654 V=800.0 PL=0
MOVL C01655 V=800.0 PL=0
MOVL C01656 V=800.0 PL=0
MOVL C01657 V=800.0 PL=0
MOVL C01658 V=800.0 PL=0
MOVL C01659 V=800.0 PL=0
MOVL C01660 V=800.0 PL=0
MOVL C01661 V=800.0 PL=0
MOVL C01662 V=800.0 PL=0
MOVL C01663 V=800.0 PL=0
MOVL C01664 V=800.0 PL=0
MOVL C01665 V=800.0 PL=0
MOVL C01666 V=800.0 PL=0
MOVL C01667 V=800.0 PL=0
MOVL C01668 V=800.0 PL=0
MOVL C01669 V=800.0 PL=0
MOVL C01670 V=800.0 PL=0
MOVL C01671 V=800.0 PL=0
MOVL C01672 V=800.0 PL=0
MOVL C01673 V=800.0 PL=0
MOVL C01674 V=800.0 PL=0
MOVL C01675 V=800.0 PL=0
MOVL C01676 V=800.0 PL=0
MOVL C01677 V=800.0 PL=0
MOVL C01678 V=800.0 PL=0
MOVL C01679 V=800.0 PL=0
MOVL C01680 V=800.0 PL=0
MOVL C01681 V=800.0 PL=0
MOVL C01682 V=800.0 PL=0
MOVL C01683 V=800.0 PL=0
MOVL C01684 V=800.0 PL=0
MOVL C01685 V=800.0 PL=0
MOVL C01686 V=800.0 PL=0
MOVL C01687 V=800.0 PL=0
MOVL C01688 V=800.0 PL=0
MOVL C01689 V=800.0 PL=0
MOVL C01690 V=800.0 PL=0
MOVL C01691 V=800.0 PL=0
MOVL C01692 V=800.0 PL=0
MOVL C01693 V=800.0 PL=0
MOVL C01694 V=800.0 PL=0
MOVL C01695 V=800.0 PL=0
MOVL C01696 V=800.0 PL=0
MOVL C01697 V=800.0 PL=0
MOVL C01698 V=800.0 PL=0
MOVL C01699 V=800.0 PL=0
MOVL C01700 V=800.0 PL=0
MOVL C01701 V=800.0 PL=0
MOVL C01702 V=800.0 PL=0
MOVL C01703 V=800.0 PL=0
MOVL C01704 V=800.0 PL=0
MOVL C01705 V=800.0 PL=0
MOVL C01706 V=800.0 PL=0
MOVL C01707 V=800.0 PL=0
MOVL C01708 V=800.0 PL=0
MOVL C01709 V=800.0 PL=0
MOVL C01710 V=800.0 PL=0
MOVL C01711 V=800.0 PL=0
MOVL C01712 V=800.0 PL=0
MOVL C01713 V=800.0 PL=0
MOVL C01714 V=800.0 PL=0
MOVL C01715 V=800.0 PL=0
MOVL C01716 V=800.0 PL=0
MOVL C01717 V=800.0 PL=0
MOVL C01718 V=800.0 PL=0
MOVL C01719 V=800.0 PL=0
MOVL C01720 V=800.0 PL=0
MOVL C01721 V=800.0 PL=0
MOVL C01722 V=800.0 PL=0
MOVL C01723 V=800.0 PL=0
MOVL C01724 V=800.0 PL=0
MOVL C01725 V=800.0 PL=0
MOVL C01726 V=800.0 PL=0
MOVL C01727 V=800.0 PL=0
MOVL C01728 V=800.0 PL=0
MOVL C01729 V=800.0 PL=0
MOVL C01730 V=800.0 PL=0
MOVL C01731 V=800.0 PL=0
MOVL C01732 V=800.0 PL=0
MOVL C01733 V=800.0 PL=0
MOVL C01734 V=800.0 PL=0
MOVL C01735 V=800.0 PL=0
MOVL C01736 V=800.0 PL=0
MOVL C01737 V=800.0 PL=0
MOVL C01738 V=800.0 PL=0
MOVL C01739 V=800.0 PL=0
MOVL C01740 V=800.0 PL=0
MOVL C01741 V=800.0 PL=0
MOVL C01742 V=800.0 PL=0
MOVL C01743 V=800.0 PL=0
MOVL C01744 V=800.0 PL=0
MOVL C01745 V=800.0 PL=0
MOVL C01746 V=800.0 PL=0
MOVL C01747 V=800.0 PL=0
MOVL C01748 V=800.0 PL=0
MOVL C01749 V=800.0 PL=0
MOVL C01750 V=800.0 PL=0
MOVL C01751 V=800.0 PL=0
MOVL C01752 V=800.0 PL=0
MOVL C01753 V=800.0 PL=0
MOVL C01754 V=800.0 PL=0
MOVL C01755 V=800.0 PL=0
MOVL C01756 V=800.0 PL=0
MOVL C01757 V=800.0 PL=0
MOVL C01758 V=800.0 PL=0
MOVL C01759 V=800.0 PL=0
MOVL C01760 V=800.0 PL=0
MOVL C01761 V=800.0 PL=0
MOVL C01762 V=800.0 PL=0
MOVL C01763 V=800.0 PL=0
MOVL C01764 V=800.0 PL=0
MOVL C01765 V=800.0 PL=0
MOVL C01766 V=800.0 PL=0
MOVL C01767 V=800.0 PL=0
MOVL C01768 V=800.0 PL=0
MOVL C01769 V=800.0 PL=0
MOVL C01770 V=800.0 PL=0
MOVL C01771 V=800.0 PL=0
MOVL C01772 V=800.0 PL=0
MOVL C01773 V=800.0 PL=0
MOVL C01774 V=800.0 PL=0
MOVL C01775 V=800.0 PL=0
MOVL C01776 V=800.0 PL=0
MOVL C01777 V=800.0 PL=0
MOVL C01778 V=800.0 PL=0
MOVL C01779 V=800.0 PL=0
MOVL C01780 V=800.0 PL=0
MOVL C01781 V=800.0 PL=0
MOVL C01782 V=800.0 PL=0
MOVL C01783 V=800.0 PL=0
MOVL C01784 V=800.0 PL=0
MOVL C01785 V=800.0 PL=0
MOVL C01786 V=800.0 PL=0
MOVL C01787 V=800.0 PL=0
MOVL C01788 V=800.0 PL=0
MOVL C01789 V=800.0 PL=0
MOVL C01790 V=800.0 PL=0
MOVL C01791 V=800.0 PL=0
MOVL C01792 V=800.0 PL=0
MOVL C01793 V=800.0 PL=0
MOVL C01794 V=800.0 PL=0
MOVL C01795 V=800.0 PL=0
MOVL C01796 V=800.0 PL=0
MOVL C01797 V=800.0 PL=0
MOVL C01798 V=800.0 PL=0
MOVL C01799 V=800.0 PL=0
MOVL C01800 V=800.0 PL=0
MOVL C01801 V=800.0 PL=0
MOVL C01802 V=800.0 PL=0
MOVL C01803 V=800.0 PL=0
MOVL C01804 V=800.0 PL=0
MOVL C01805 V=800.0 PL=0
MOVL C01806 V=800.0 PL=0
MOVL C01807 V=800.0 PL=0
MOVL C01808 V=800.0 PL=0
MOVL C01809 V=800.0 PL=0
MOVL C01810 V=800.0 PL=0
MOVL C01811 V=800.0 PL=0
MOVL C01812 V=800.0 PL=0
MOVL C01813 V=800.0 PL=0
MOVL C01814 V=800.0 PL=0
MOVL C01815 V=800.0 PL=0
MOVL C01816 V=800.0 PL=0
MOVL C01817 V=800.0 PL=0
MOVL C01818 V=800.0 PL=0
MOVL C01819 V=800.0 PL=0
MOVL C01820 V=800.0 PL=0
MOVL C01821 V=800.0 PL=0
MOVL C01822 V=800.0 PL=0
MOVL C01823 V=800.0 PL=0
MOVL C01824 V=800.0 PL=0
MOVL C01825 V=800.0 PL=0
MOVL C01826 V=800.0 PL=0
MOVL C01827 V=800.0 PL=0
MOVL C01828 V=800.0 PL=0
MOVL C01829 V=800.0 PL=0
MOVL C01830 V=800.0 PL=0
MOVL C01831 V=800.0 PL=0
MOVL C01832 V=800.0 PL=0
MOVL C01833 V=800.0 PL=0
MOVL C01834 V=800.0 PL=0
MOVL C01835 V=800.0 PL=0
MOVL C01836 V=800.0 PL=0
MOVL C01837 V=800.0 PL=0
MOVL C01838 V=800.0 PL=0
MOVL C01839 V=800.0 PL=0
MOVL C01840 V=800.0 PL=0
MOVL C01841 V=800.0 PL=0
MOVL C01842 V=800.0 PL=0
MOVL C01843 V=800.0 PL=0
MOVL C01844 V=800.0 PL=0
MOVL C01845 V=800.0 PL=0
MOVL C01846 V=800.0 PL=0
MOVL C01847 V=800.0 PL=0
MOVL C01848 V=800.0 PL=0
MOVL C01849 V=800.0 PL=0
MOVL C01850 V=800.0 PL=0
MOVL C01851 V=800.0 PL=0
MOVL C01852 V=800.0 PL=0
MOVL C01853 V=800.0 PL=0
MOVL C01854 V=800.0 PL=0
MOVL C01855 V=800.0 PL=0
MOVL C01856 V=800.0 PL=0
MOVL C01857 V=800.0 PL=0
MOVL C01858 V=800.0 PL=0
MOVL C01859 V=800.0 PL=0
MOVL C01860 V=800.0 PL=0
MOVL C01861 V=800.0 PL=0
MOVL C01862 V=800.0 PL=0
MOVL C01863 V=800.0 PL=0
MOVL C01864 V=800.0 PL=0
MOVL C01865 V=800.0 PL=0
MOVL C01866 V=800.0 PL=0
MOVL C01867 V=800.0 PL=0
MOVL C01868 V=800.0 PL=0
MOVL C01869 V=800.0 PL=0
MOVL C01870 V=800.0 PL=0
MOVL C01871 V=800.0 PL=0
MOVL C01872 V=800.0 PL=0
MOVL C01873 V=800.0 PL=0
MOVL C01874 V=800.0 PL=0
MOVL C01875 V=800.0 PL=0
MOVL C01876 V=800.0 PL=0
MOVL C01877 V=800.0 PL=0
MOVL C01878 V=800.0 PL=0
MOVL C01879 V=800.0 PL=0
MOVL C01880 V=800.0 PL=0
MOVL C01881 V=800.0 PL=0
MOVL C01882 V=800.0 PL=0
MOVL C01883 V=800.0 PL=0
MOVL C01884 V=800.0 PL=0
MOVL C01885 V=800.0 PL=0
MOVL C01886 V=800.0 PL=0
MOVL C01887 V=800.0 PL=0
MOVL C01888 V=800.0 PL=0
MOVL C01889 V=800.0 PL=0
MOVL C01890 V=800.0 PL=0
MOVL C01891 V=800.0 PL=0
MOVL C01892 V=800.0 PL=0
MOVL C01893 V=800.0 PL=0
MOVL C01894 V=800.0 PL=0
MOVL C01895 V=800.0 PL=0
MOVL C01896 V=800.0 PL=0
MOVL C01897 V=800.0 PL=0
MOVL C01898 V=800.0 PL=0
MOVL C01899 V=800.0 PL=0
MOVL C01900 V=800.0 PL=0
MOVL C01901 V=800.0 PL=0
MOVL C01902 V=800.0 PL=0
MOVL C01903 V=800.0 PL=0
MOVL C01904 V=800.0 PL=0
MOVL C01905 V=800.0 PL=0
MOVL C01906 V=800.0 PL=0
MOVL C01907 V=800.0 PL=0
MOVL C01908 V=800.0 PL=0
MOVL C01909 V=800.0 PL=0
MOVL C01910 V=800.0 PL=0
MOVL C01911 V=800.0 PL=0
MOVL C01912 V=800.0 PL=0
MOVL C01913 V=800.0 PL=0
MOVL C01914 V=800.0 PL=0
MOVL C01915 V=800.0 PL=0
MOVL C01916 V=800.0 PL=0
MOVL C01917 V=800.0 PL=0
MOVL C01918 V=800.0 PL=0
MOVL C01919 V=800.0 PL=0
MOVL C01920 V=800.0 PL=0
MOVL C01921 V=800.0 PL=0
MOVL C01922 V=800.0 PL=0
MOVL C01923 V=800.0 PL=0
MOVL C01924 V=800.0 PL=0
MOVL C01925 V=800.0 PL=0
MOVL C01926 V=800.0 PL=0
MOVL C01927 V=800.0 PL=0
MOVL C01928 V=800.0 PL=0
MOVL C01929 V=800.0 PL=0
MOVL C01930 V=800.0 PL=0
MOVL C01931 V=800.0 PL=0
MOVL C01932 V=800.0 PL=0
MOVL C01933 V=800.0 PL=0
MOVL C01934 V=800.0 PL=0
MOVL C01935 V=800.0 PL=0
MOVL C01936 V=800.0 PL=0
MOVL C01937 V=800.0 PL=0
MOVL C01938 V=800.0 PL=0
MOVL C01939 V=800.0 PL=0
MOVL C01940 V=800.0 PL=0
MOVL C01941 V=800.0 PL=0
MOVL C01942 V=800.0 PL=0
MOVL C01943 V=800.0 PL=0
MOVL C01944 V=800.0 PL=0
MOVL C01945 V=800.0 PL=0
MOVL C01946 V=800.0 PL=0
MOVL C01947 V=800.0 PL=0
MOVL C01948 V=800.0 PL=0
MOVL C01949 V=800.0 PL=0
MOVL C01950 V=800.0 PL=0
MOVL C01951 V=800.0 PL=0
MOVL C01952 V=800.0 PL=0
MOVL C01953 V=800.0 PL=0
MOVL C01954 V=800.0 PL=0
MOVL C01955 V=800.0 PL=0
